Page_410_WorkStation_Axis3;
Page_420_WorkStation_ToolDia;
Page_430_WorkStation_Prism;
Page_460_WorkStation_ErrorList;
Page_470_WorkStation_Parameter3;
END_FUNCTION_BLOCK
ACTION Page_000_Start:
(* QVis page 0, start page *)
iIndexPage:=0;
iPageNumber:=iPageNumber+1;
T_Visu.T_PageIndex[iIndexPage].iIndexConfigPage:=iPageNumber;
ptrConfigPage:=ADR(T_Visu.T_ConfigPage[T_Visu.T_PageIndex[iIndexPage].iIndexConfigPage]);
ptrConfigPage^.sName:='Start page';
ptrConfigPage^.wMaskBtPanelLeft:=16#0;
ptrConfigPage^.wMaskBtPanelRight:=16#0;
ptrConfigPage^.wMaskFunctionPanel:=16#0;
(* Navigation panel restriction *)
ptrConfigPage^.wMaskTouchScreenNavPanel:=16#0;
(* Active machine movement mask *)
ptrConfigPage^.wMaskActiveMachineBtPanelLeft:=16#0;
ptrConfigPage^.wMaskActiveMachineBtPanelRight:=16#0;
ptrConfigPage^.wMaskActiveMachineFunctionPanel:=16#0;
ptrConfigPage^.wMaskActiveMachineNavPanel:=16#0;
(* Button edge action *)
ptrConfigPage^.aiRTrigActionPanelRight[1]:=0;
ptrConfigPage^.aiRTrigActionPanelRight[2]:=0;
ptrConfigPage^.aiRTrigActionPanelRight[3]:=0;
ptrConfigPage^.aiRTrigActionPanelRight[4]:=0;
ptrConfigPage^.aiRTrigActionPanelRight[5]:=0;
ptrConfigPage^.aiFTrigActionPanelRight[1]:=0;
ptrConfigPage^.aiFTrigActionPanelRight[2]:=0;
ptrConfigPage^.aiFTrigActionPanelRight[3]:=0;
ptrConfigPage^.aiFTrigActionPanelRight[4]:=0;
ptrConfigPage^.aiFTrigActionPanelRight[5]:=0;
ptrConfigPage^.aiDelayActionPanelRight[1]:=0;
ptrConfigPage^.aiDelayActionPanelRight[2]:=0;
ptrConfigPage^.aiDelayActionPanelRight[3]:=0;
ptrConfigPage^.aiDelayActionPanelRight[4]:=0;
ptrConfigPage^.aiDelayActionPanelRight[5]:=0;
ptrConfigPage^.aiRTrigActionFunctionPanel[1]:=0;
ptrConfigPage^.aiRTrigActionFunctionPanel[2]:=0;
ptrConfigPage^.aiRTrigActionFunctionPanel[3]:=0;
ptrConfigPage^.aiRTrigActionFunctionPanel[4]:=0;
ptrConfigPage^.aiRTrigActionFunctionPanel[5]:=0;
ptrConfigPage^.aiRTrigActionFunctionPanel[6]:=0;
ptrConfigPage^.aiRTrigActionFunctionPanel[7]:=0;
ptrConfigPage^.aiRTrigActionFunctionPanel[8]:=0;
ptrConfigPage^.aiRTrigActionFunctionPanel[9]:=0;
ptrConfigPage^.aiRTrigActionFunctionPanel[10]:=0;
ptrConfigPage^.aiRTrigActionFunctionPanel[11]:=0;
ptrConfigPage^.aiRTrigActionFunctionPanel[12]:=0;
ptrConfigPage^.aiFTrigActionTouchScreenNavPanel[1]:=0;
ptrConfigPage^.aiFTrigActionTouchScreenNavPanel[2]:=0;
ptrConfigPage^.aiFTrigActionTouchScreenNavPanel[3]:=0;
ptrConfigPage^.aiFTrigActionTouchScreenNavPanel[4]:=0;
ptrConfigPage^.aiFTrigActionTouchScreenNavPanel[5]:=0;
ptrConfigPage^.aiFTrigActionTouchScreenNavPanel[6]:=0;
ptrConfigPage^.xMaskBtStart:=TRUE;
ptrConfigPage^.xMaskBtStop:=FALSE;
END_ACTION
ACTION Page_001_BIOS:
(* QVis page 1, BIOS Password StartUp *)
iIndexPage:=1;
iPageNumber:=iPageNumber+1;
T_Visu.T_PageIndex[iIndexPage].iIndexConfigPage:=iPageNumber;
ptrConfigPage:=ADR(T_Visu.T_ConfigPage[T_Visu.T_PageIndex[iIndexPage].iIndexConfigPage]);
ptrConfigPage^.sName:='BIOS Password StartUp';
ptrConfigPage^.wMaskBtPanelLeft:=16#0;
ptrConfigPage^.wMaskBtPanelRight:=16#0;
ptrConfigPage^.wMaskFunctionPanel:=16#0;
(* Navigation panel restriction *)
ptrConfigPage^.wMaskTouchScreenNavPanel:=16#0;
(* Active machine movement mask *)
ptrConfigPage^.wMaskActiveMachineBtPanelLeft:=16#0;
ptrConfigPage^.wMaskActiveMachineBtPanelRight:=16#0;
ptrConfigPage^.wMaskActiveMachineFunctionPanel:=16#0;
ptrConfigPage^.wMaskActiveMachineNavPanel:=16#0;
(* Button edge action *)
ptrConfigPage^.aiRTrigActionPanelRight[1]:=0;
ptrConfigPage^.aiRTrigActionPanelRight[2]:=0;
ptrConfigPage^.aiRTrigActionPanelRight[3]:=0;
ptrConfigPage^.aiRTrigActionPanelRight[4]:=0;
ptrConfigPage^.aiRTrigActionPanelRight[5]:=0;
ptrConfigPage^.aiFTrigActionPanelRight[1]:=0;
ptrConfigPage^.aiFTrigActionPanelRight[2]:=0;
ptrConfigPage^.aiFTrigActionPanelRight[3]:=0;
ptrConfigPage^.aiFTrigActionPanelRight[4]:=0;
ptrConfigPage^.aiFTrigActionPanelRight[5]:=0;
ptrConfigPage^.aiDelayActionPanelRight[1]:=0;
ptrConfigPage^.aiDelayActionPanelRight[2]:=0;
ptrConfigPage^.aiDelayActionPanelRight[3]:=0;
ptrConfigPage^.aiDelayActionPanelRight[4]:=0;
ptrConfigPage^.aiDelayActionPanelRight[5]:=0;
ptrConfigPage^.aiRTrigActionFunctionPanel[1]:=0;
ptrConfigPage^.aiRTrigActionFunctionPanel[2]:=0;
ptrConfigPage^.aiRTrigActionFunctionPanel[3]:=0;
ptrConfigPage^.aiRTrigActionFunctionPanel[4]:=0;
ptrConfigPage^.aiRTrigActionFunctionPanel[5]:=0;
ptrConfigPage^.aiRTrigActionFunctionPanel[6]:=0;
ptrConfigPage^.aiRTrigActionFunctionPanel[7]:=0;
ptrConfigPage^.aiRTrigActionFunctionPanel[8]:=0;
ptrConfigPage^.aiRTrigActionFunctionPanel[9]:=0;
ptrConfigPage^.aiRTrigActionFunctionPanel[10]:=0;
ptrConfigPage^.aiRTrigActionFunctionPanel[11]:=0;
ptrConfigPage^.aiRTrigActionFunctionPanel[12]:=0;
ptrConfigPage^.aiFTrigActionTouchScreenNavPanel[1]:=0;
ptrConfigPage^.aiFTrigActionTouchScreenNavPanel[2]:=0;
ptrConfigPage^.aiFTrigActionTouchScreenNavPanel[3]:=0;
ptrConfigPage^.aiFTrigActionTouchScreenNavPanel[4]:=0;
ptrConfigPage^.aiFTrigActionTouchScreenNavPanel[5]:=0;
ptrConfigPage^.aiFTrigActionTouchScreenNavPanel[6]:=0;
ptrConfigPage^.xMaskBtStart:=FALSE;
ptrConfigPage^.xMaskBtStop:=FALSE;
END_ACTION
ACTION Page_002_BIOS:
(* QVis page 2, BIOS Parameter StartUp *)
iIndexPage:=2;
iPageNumber:=iPageNumber+1;
T_Visu.T_PageIndex[iIndexPage].iIndexConfigPage:=iPageNumber;
ptrConfigPage:=ADR(T_Visu.T_ConfigPage[T_Visu.T_PageIndex[iIndexPage].iIndexConfigPage]);
ptrConfigPage^.sName:='BIOS Parameter StartUp';
ptrConfigPage^.wMaskBtPanelLeft:=16#0;
ptrConfigPage^.wMaskBtPanelRight:=16#200;
ptrConfigPage^.wMaskFunctionPanel:=16#0;
(* Navigation panel restriction *)
ptrConfigPage^.wMaskTouchScreenNavPanel:=16#0;
(* Active machine movement mask *)
ptrConfigPage^.wMaskActiveMachineBtPanelLeft:=16#0;
ptrConfigPage^.wMaskActiveMachineBtPanelRight:=16#200;
ptrConfigPage^.wMaskActiveMachineFunctionPanel:=16#0;
ptrConfigPage^.wMaskActiveMachineNavPanel:=16#0;
(* Button edge action *)
ptrConfigPage^.aiRTrigActionPanelRight[1]:=0;
ptrConfigPage^.aiRTrigActionPanelRight[2]:=0;
ptrConfigPage^.aiRTrigActionPanelRight[3]:=0;
ptrConfigPage^.aiRTrigActionPanelRight[4]:=0;
ptrConfigPage^.aiRTrigActionPanelRight[5]:=0;
ptrConfigPage^.aiFTrigActionPanelRight[1]:=0;
ptrConfigPage^.aiFTrigActionPanelRight[2]:=0;
ptrConfigPage^.aiFTrigActionPanelRight[3]:=0;
ptrConfigPage^.aiFTrigActionPanelRight[4]:=0;
ptrConfigPage^.aiFTrigActionPanelRight[5]:=0;
ptrConfigPage^.aiDelayActionPanelRight[1]:=0;
ptrConfigPage^.aiDelayActionPanelRight[2]:=0;
ptrConfigPage^.aiDelayActionPanelRight[3]:=0;
ptrConfigPage^.aiDelayActionPanelRight[4]:=0;
ptrConfigPage^.aiDelayActionPanelRight[5]:=0;
ptrConfigPage^.aiRTrigActionFunctionPanel[1]:=0;
ptrConfigPage^.aiRTrigActionFunctionPanel[2]:=0;
ptrConfigPage^.aiRTrigActionFunctionPanel[3]:=0;
ptrConfigPage^.aiRTrigActionFunctionPanel[4]:=0;
ptrConfigPage^.aiRTrigActionFunctionPanel[5]:=0;
ptrConfigPage^.aiRTrigActionFunctionPanel[6]:=0;
ptrConfigPage^.aiRTrigActionFunctionPanel[7]:=0;
ptrConfigPage^.aiRTrigActionFunctionPanel[8]:=0;
ptrConfigPage^.aiRTrigActionFunctionPanel[9]:=0;
ptrConfigPage^.aiRTrigActionFunctionPanel[10]:=0;
ptrConfigPage^.aiRTrigActionFunctionPanel[11]:=0;
ptrConfigPage^.aiRTrigActionFunctionPanel[12]:=0;
ptrConfigPage^.aiFTrigActionTouchScreenNavPanel[1]:=0;
ptrConfigPage^.aiFTrigActionTouchScreenNavPanel[2]:=0;
ptrConfigPage^.aiFTrigActionTouchScreenNavPanel[3]:=0;
ptrConfigPage^.aiFTrigActionTouchScreenNavPanel[4]:=0;
ptrConfigPage^.aiFTrigActionTouchScreenNavPanel[5]:=0;
ptrConfigPage^.aiFTrigActionTouchScreenNavPanel[6]:=0;
ptrConfigPage^.xMaskBtStart:=FALSE;
ptrConfigPage^.xMaskBtStop:=FALSE;
END_ACTION
ACTION Page_010_Auto_Geometry1:
(* QVis page 10, Auto Geometry, page 1 *)
iIndexPage:=10;
iPageNumber:=iPageNumber+1;
T_Visu.T_PageIndex[iIndexPage].iIndexConfigPage:=iPageNumber;
ptrConfigPage:=ADR(T_Visu.T_ConfigPage[T_Visu.T_PageIndex[iIndexPage].iIndexConfigPage]);
ptrConfigPage^.sName:='Auto Geometry, page 1';
ptrConfigPage^.wMaskBtPanelLeft:=16#F;
ptrConfigPage^.wMaskBtPanelRight:=16#200;
(*08.07.2014: KFS	{	*)
(*ptrConfigPage^.wMaskFunctionPanel:=16#F;*)
ptrConfigPage^.wMaskFunctionPanel:=16#3F;
(*08.07.2014: KFS	}	*)
(* Navigation panel restriction *)
ptrConfigPage^.wMaskTouchScreenNavPanel:=16#3F;
(* Active machine movement mask *)
ptrConfigPage^.wMaskActiveMachineBtPanelLeft:=16#F;
ptrConfigPage^.wMaskActiveMachineBtPanelRight:=16#220;
ptrConfigPage^.wMaskActiveMachineFunctionPanel:=16#0;
ptrConfigPage^.wMaskActiveMachineNavPanel:=16#3F;
(* Button edge action *)
ptrConfigPage^.aiRTrigActionPanelRight[1]:=801;
ptrConfigPage^.aiRTrigActionPanelRight[2]:=0;
ptrConfigPage^.aiRTrigActionPanelRight[3]:=0;
ptrConfigPage^.aiRTrigActionPanelRight[4]:=0;
ptrConfigPage^.aiRTrigActionPanelRight[5]:=12;
ptrConfigPage^.aiFTrigActionPanelRight[1]:=0;
ptrConfigPage^.aiFTrigActionPanelRight[2]:=0;
ptrConfigPage^.aiFTrigActionPanelRight[3]:=0;
ptrConfigPage^.aiFTrigActionPanelRight[4]:=0;
ptrConfigPage^.aiFTrigActionPanelRight[5]:=0;
ptrConfigPage^.aiDelayActionPanelRight[1]:=0;
ptrConfigPage^.aiDelayActionPanelRight[2]:=0;
ptrConfigPage^.aiDelayActionPanelRight[3]:=0;
ptrConfigPage^.aiDelayActionPanelRight[4]:=0;
ptrConfigPage^.aiDelayActionPanelRight[5]:=0;
ptrConfigPage^.aiRTrigActionFunctionPanel[1]:=102;
ptrConfigPage^.aiRTrigActionFunctionPanel[2]:=103;
ptrConfigPage^.aiRTrigActionFunctionPanel[3]:=501;
ptrConfigPage^.aiRTrigActionFunctionPanel[4]:=106;
ptrConfigPage^.aiRTrigActionFunctionPanel[5]:=107;
ptrConfigPage^.aiRTrigActionFunctionPanel[6]:=108;
ptrConfigPage^.aiRTrigActionFunctionPanel[7]:=0;
ptrConfigPage^.aiRTrigActionFunctionPanel[8]:=0;
ptrConfigPage^.aiRTrigActionFunctionPanel[9]:=0;
ptrConfigPage^.aiRTrigActionFunctionPanel[10]:=0;
ptrConfigPage^.aiRTrigActionFunctionPanel[11]:=0;
ptrConfigPage^.aiRTrigActionFunctionPanel[12]:=0;
ptrConfigPage^.aiFTrigActionTouchScreenNavPanel[1]:=10010;
ptrConfigPage^.aiFTrigActionTouchScreenNavPanel[2]:=10020;
ptrConfigPage^.aiFTrigActionTouchScreenNavPanel[3]:=10030;
ptrConfigPage^.aiFTrigActionTouchScreenNavPanel[4]:=10040;
ptrConfigPage^.aiFTrigActionTouchScreenNavPanel[5]:=10050;
ptrConfigPage^.aiFTrigActionTouchScreenNavPanel[6]:=10060;
ptrConfigPage^.xMaskBtStart:=TRUE;
ptrConfigPage^.xMaskBtStop:=TRUE;
END_ACTION
ACTION Page_011_Auto_Geometry2:
(* QVis page 11, Auto Geometry, page 2 *)
iIndexPage:=11;
iPageNumber:=iPageNumber+1;
T_Visu.T_PageIndex[iIndexPage].iIndexConfigPage:=iPageNumber;
ptrConfigPage:=ADR(T_Visu.T_ConfigPage[T_Visu.T_PageIndex[iIndexPage].iIndexConfigPage]);
ptrConfigPage^.sName:='Auto Geometry, page 2';
ptrConfigPage^.wMaskBtPanelLeft:=16#F;
ptrConfigPage^.wMaskBtPanelRight:=16#200;
ptrConfigPage^.wMaskFunctionPanel:=16#EF;
(* Navigation panel restriction *)
ptrConfigPage^.wMaskTouchScreenNavPanel:=16#3F;
(* Active machine movement mask *)
ptrConfigPage^.wMaskActiveMachineBtPanelLeft:=16#0;
ptrConfigPage^.wMaskActiveMachineBtPanelRight:=16#0;
ptrConfigPage^.wMaskActiveMachineFunctionPanel:=16#0;
ptrConfigPage^.wMaskActiveMachineNavPanel:=16#3F;
(* Button edge action *)
ptrConfigPage^.aiRTrigActionPanelRight[1]:=0;
ptrConfigPage^.aiRTrigActionPanelRight[2]:=0;
ptrConfigPage^.aiRTrigActionPanelRight[3]:=0;
ptrConfigPage^.aiRTrigActionPanelRight[4]:=0;
ptrConfigPage^.aiRTrigActionPanelRight[5]:=12;
ptrConfigPage^.aiFTrigActionPanelRight[1]:=0;
ptrConfigPage^.aiFTrigActionPanelRight[2]:=0;
ptrConfigPage^.aiFTrigActionPanelRight[3]:=0;
ptrConfigPage^.aiFTrigActionPanelRight[4]:=0;
ptrConfigPage^.aiFTrigActionPanelRight[5]:=0;
ptrConfigPage^.aiDelayActionPanelRight[1]:=0;
ptrConfigPage^.aiDelayActionPanelRight[2]:=0;
ptrConfigPage^.aiDelayActionPanelRight[3]:=0;
ptrConfigPage^.aiDelayActionPanelRight[4]:=0;
ptrConfigPage^.aiDelayActionPanelRight[5]:=0;
ptrConfigPage^.aiRTrigActionFunctionPanel[1]:=110;
ptrConfigPage^.aiRTrigActionFunctionPanel[2]:=111;
ptrConfigPage^.aiRTrigActionFunctionPanel[3]:=114;
ptrConfigPage^.aiRTrigActionFunctionPanel[4]:=115;
ptrConfigPage^.aiRTrigActionFunctionPanel[5]:=0;
ptrConfigPage^.aiRTrigActionFunctionPanel[6]:=116;
ptrConfigPage^.aiRTrigActionFunctionPanel[7]:=112;
ptrConfigPage^.aiRTrigActionFunctionPanel[8]:=113;
ptrConfigPage^.aiRTrigActionFunctionPanel[9]:=0;
ptrConfigPage^.aiRTrigActionFunctionPanel[10]:=0;
ptrConfigPage^.aiRTrigActionFunctionPanel[11]:=0;
ptrConfigPage^.aiRTrigActionFunctionPanel[12]:=0;
ptrConfigPage^.aiFTrigActionTouchScreenNavPanel[1]:=10010;
ptrConfigPage^.aiFTrigActionTouchScreenNavPanel[2]:=10020;
ptrConfigPage^.aiFTrigActionTouchScreenNavPanel[3]:=10030;
ptrConfigPage^.aiFTrigActionTouchScreenNavPanel[4]:=10040;
ptrConfigPage^.aiFTrigActionTouchScreenNavPanel[5]:=10050;
ptrConfigPage^.aiFTrigActionTouchScreenNavPanel[6]:=10060;
ptrConfigPage^.xMaskBtStart:=TRUE;
ptrConfigPage^.xMaskBtStop:=TRUE;
END_ACTION
ACTION Page_020_Auto_Groove1:
(* QVis page 20, Auto Groove, page 1 *)
iIndexPage:=20;
iPageNumber:=iPageNumber+1;
T_Visu.T_PageIndex[iIndexPage].iIndexConfigPage:=iPageNumber;
ptrConfigPage:=ADR(T_Visu.T_ConfigPage[T_Visu.T_PageIndex[iIndexPage].iIndexConfigPage]);
ptrConfigPage^.sName:='Auto Groove, page 1';
ptrConfigPage^.wMaskBtPanelLeft:=16#F;
ptrConfigPage^.wMaskBtPanelRight:=16#200;
ptrConfigPage^.wMaskFunctionPanel:=16#3F;
(* Navigation panel restriction *)
ptrConfigPage^.wMaskTouchScreenNavPanel:=16#3F;
(* Active machine movement mask *)
ptrConfigPage^.wMaskActiveMachineBtPanelLeft:=16#F;
ptrConfigPage^.wMaskActiveMachineBtPanelRight:=16#200;
ptrConfigPage^.wMaskActiveMachineFunctionPanel:=16#0;
ptrConfigPage^.wMaskActiveMachineNavPanel:=16#3F;
(* Button edge action *)
ptrConfigPage^.aiRTrigActionPanelRight[1]:=0;
ptrConfigPage^.aiRTrigActionPanelRight[2]:=0;
ptrConfigPage^.aiRTrigActionPanelRight[3]:=0;
ptrConfigPage^.aiRTrigActionPanelRight[4]:=0;
ptrConfigPage^.aiRTrigActionPanelRight[5]:=12;
ptrConfigPage^.aiFTrigActionPanelRight[1]:=0;
ptrConfigPage^.aiFTrigActionPanelRight[2]:=0;
ptrConfigPage^.aiFTrigActionPanelRight[3]:=0;
ptrConfigPage^.aiFTrigActionPanelRight[4]:=0;
ptrConfigPage^.aiFTrigActionPanelRight[5]:=0;
ptrConfigPage^.aiDelayActionPanelRight[1]:=0;
ptrConfigPage^.aiDelayActionPanelRight[2]:=0;
ptrConfigPage^.aiDelayActionPanelRight[3]:=0;
ptrConfigPage^.aiDelayActionPanelRight[4]:=0;
ptrConfigPage^.aiDelayActionPanelRight[5]:=0;
ptrConfigPage^.aiRTrigActionFunctionPanel[1]:=102;
ptrConfigPage^.aiRTrigActionFunctionPanel[2]:=103;
ptrConfigPage^.aiRTrigActionFunctionPanel[3]:=501;
ptrConfigPage^.aiRTrigActionFunctionPanel[4]:=105;
ptrConfigPage^.aiRTrigActionFunctionPanel[5]:=107;
ptrConfigPage^.aiRTrigActionFunctionPanel[6]:=104;
ptrConfigPage^.aiRTrigActionFunctionPanel[7]:=0;
ptrConfigPage^.aiRTrigActionFunctionPanel[8]:=0;
ptrConfigPage^.aiRTrigActionFunctionPanel[9]:=0;
ptrConfigPage^.aiRTrigActionFunctionPanel[10]:=0;
ptrConfigPage^.aiRTrigActionFunctionPanel[11]:=0;
ptrConfigPage^.aiRTrigActionFunctionPanel[12]:=0;
ptrConfigPage^.aiFTrigActionTouchScreenNavPanel[1]:=10010;
ptrConfigPage^.aiFTrigActionTouchScreenNavPanel[2]:=10020;
ptrConfigPage^.aiFTrigActionTouchScreenNavPanel[3]:=10030;
ptrConfigPage^.aiFTrigActionTouchScreenNavPanel[4]:=10040;
ptrConfigPage^.aiFTrigActionTouchScreenNavPanel[5]:=10050;
ptrConfigPage^.aiFTrigActionTouchScreenNavPanel[6]:=10060;
ptrConfigPage^.xMaskBtStart:=TRUE;
ptrConfigPage^.xMaskBtStop:=TRUE;
END_ACTION
ACTION Page_021_Auto_Groove2:
(* QVis page 21, Auto Groove, page 2 *)
iIndexPage:=21;
iPageNumber:=iPageNumber+1;
T_Visu.T_PageIndex[iIndexPage].iIndexConfigPage:=iPageNumber;
ptrConfigPage:=ADR(T_Visu.T_ConfigPage[T_Visu.T_PageIndex[iIndexPage].iIndexConfigPage]);
ptrConfigPage^.sName:='Auto Groove, page 2';
ptrConfigPage^.wMaskBtPanelLeft:=16#F;
ptrConfigPage^.wMaskBtPanelRight:=16#200;
ptrConfigPage^.wMaskFunctionPanel:=16#EF;
(* Navigation panel restriction *)
ptrConfigPage^.wMaskTouchScreenNavPanel:=16#3F;
(* Active machine movement mask *)
ptrConfigPage^.wMaskActiveMachineBtPanelLeft:=16#0;
ptrConfigPage^.wMaskActiveMachineBtPanelRight:=16#0;
ptrConfigPage^.wMaskActiveMachineFunctionPanel:=16#0;
ptrConfigPage^.wMaskActiveMachineNavPanel:=16#3F;
(* Button edge action *)
ptrConfigPage^.aiRTrigActionPanelRight[1]:=0;
ptrConfigPage^.aiRTrigActionPanelRight[2]:=0;
ptrConfigPage^.aiRTrigActionPanelRight[3]:=0;
ptrConfigPage^.aiRTrigActionPanelRight[4]:=0;
ptrConfigPage^.aiRTrigActionPanelRight[5]:=12;
ptrConfigPage^.aiFTrigActionPanelRight[1]:=0;
ptrConfigPage^.aiFTrigActionPanelRight[2]:=0;
ptrConfigPage^.aiFTrigActionPanelRight[3]:=0;
ptrConfigPage^.aiFTrigActionPanelRight[4]:=0;
ptrConfigPage^.aiFTrigActionPanelRight[5]:=0;
ptrConfigPage^.aiDelayActionPanelRight[1]:=0;
ptrConfigPage^.aiDelayActionPanelRight[2]:=0;
ptrConfigPage^.aiDelayActionPanelRight[3]:=0;
ptrConfigPage^.aiDelayActionPanelRight[4]:=0;
ptrConfigPage^.aiDelayActionPanelRight[5]:=0;
ptrConfigPage^.aiRTrigActionFunctionPanel[1]:=110;
ptrConfigPage^.aiRTrigActionFunctionPanel[2]:=111;
ptrConfigPage^.aiRTrigActionFunctionPanel[3]:=114;
ptrConfigPage^.aiRTrigActionFunctionPanel[4]:=115;
ptrConfigPage^.aiRTrigActionFunctionPanel[5]:=0;
ptrConfigPage^.aiRTrigActionFunctionPanel[6]:=116;
ptrConfigPage^.aiRTrigActionFunctionPanel[7]:=112;
ptrConfigPage^.aiRTrigActionFunctionPanel[8]:=113;
ptrConfigPage^.aiRTrigActionFunctionPanel[9]:=0;
ptrConfigPage^.aiRTrigActionFunctionPanel[10]:=0;
ptrConfigPage^.aiRTrigActionFunctionPanel[11]:=0;
ptrConfigPage^.aiRTrigActionFunctionPanel[12]:=0;
ptrConfigPage^.aiFTrigActionTouchScreenNavPanel[1]:=10010;
ptrConfigPage^.aiFTrigActionTouchScreenNavPanel[2]:=10020;
ptrConfigPage^.aiFTrigActionTouchScreenNavPanel[3]:=10030;
ptrConfigPage^.aiFTrigActionTouchScreenNavPanel[4]:=10040;
ptrConfigPage^.aiFTrigActionTouchScreenNavPanel[5]:=10050;
ptrConfigPage^.aiFTrigActionTouchScreenNavPanel[6]:=10060;
ptrConfigPage^.xMaskBtStart:=TRUE;
ptrConfigPage^.xMaskBtStop:=TRUE;
END_ACTION
ACTION Page_030_Auto_Reference:
(* QVis page 30, Reference *)
iIndexPage:=30;
iPageNumber:=iPageNumber+1;
T_Visu.T_PageIndex[iIndexPage].iIndexConfigPage:=iPageNumber;
ptrConfigPage:=ADR(T_Visu.T_ConfigPage[T_Visu.T_PageIndex[iIndexPage].iIndexConfigPage]);
ptrConfigPage^.sName:='Reference';
ptrConfigPage^.wMaskBtPanelLeft:=16#F;
ptrConfigPage^.wMaskBtPanelRight:=16#1E0;
ptrConfigPage^.wMaskFunctionPanel:=16#D;
(* Navigation panel restriction *)
ptrConfigPage^.wMaskTouchScreenNavPanel:=16#3F;
(* Active machine movement mask *)
ptrConfigPage^.wMaskActiveMachineBtPanelLeft:=16#F;
ptrConfigPage^.wMaskActiveMachineBtPanelRight:=16#60;
ptrConfigPage^.wMaskActiveMachineFunctionPanel:=16#0;
ptrConfigPage^.wMaskActiveMachineNavPanel:=16#3F;
(* Button edge action *)
ptrConfigPage^.aiRTrigActionPanelRight[1]:=312;
ptrConfigPage^.aiRTrigActionPanelRight[2]:=310;
ptrConfigPage^.aiRTrigActionPanelRight[3]:=316;
ptrConfigPage^.aiRTrigActionPanelRight[4]:=314;
ptrConfigPage^.aiRTrigActionPanelRight[5]:=0;
ptrConfigPage^.aiFTrigActionPanelRight[1]:=0;
ptrConfigPage^.aiFTrigActionPanelRight[2]:=0;
ptrConfigPage^.aiFTrigActionPanelRight[3]:=301;
ptrConfigPage^.aiFTrigActionPanelRight[4]:=301;
ptrConfigPage^.aiFTrigActionPanelRight[5]:=0;
ptrConfigPage^.aiDelayActionPanelRight[1]:=0;
ptrConfigPage^.aiDelayActionPanelRight[2]:=0;
ptrConfigPage^.aiDelayActionPanelRight[3]:=0;
ptrConfigPage^.aiDelayActionPanelRight[4]:=0;
ptrConfigPage^.aiDelayActionPanelRight[5]:=0;
ptrConfigPage^.aiRTrigActionFunctionPanel[1]:=320;
ptrConfigPage^.aiRTrigActionFunctionPanel[2]:=0;
ptrConfigPage^.aiRTrigActionFunctionPanel[3]:=501;
ptrConfigPage^.aiRTrigActionFunctionPanel[4]:=106;
ptrConfigPage^.aiRTrigActionFunctionPanel[5]:=0;
ptrConfigPage^.aiRTrigActionFunctionPanel[6]:=0;
ptrConfigPage^.aiRTrigActionFunctionPanel[7]:=0;
ptrConfigPage^.aiRTrigActionFunctionPanel[8]:=0;
ptrConfigPage^.aiRTrigActionFunctionPanel[9]:=0;
ptrConfigPage^.aiRTrigActionFunctionPanel[10]:=0;
ptrConfigPage^.aiRTrigActionFunctionPanel[11]:=0;
ptrConfigPage^.aiRTrigActionFunctionPanel[12]:=0;
ptrConfigPage^.aiFTrigActionTouchScreenNavPanel[1]:=10010;
ptrConfigPage^.aiFTrigActionTouchScreenNavPanel[2]:=10020;
ptrConfigPage^.aiFTrigActionTouchScreenNavPanel[3]:=10030;
ptrConfigPage^.aiFTrigActionTouchScreenNavPanel[4]:=10040;
ptrConfigPage^.aiFTrigActionTouchScreenNavPanel[5]:=10050;
ptrConfigPage^.aiFTrigActionTouchScreenNavPanel[6]:=10060;
ptrConfigPage^.xMaskBtStart:=TRUE;
ptrConfigPage^.xMaskBtStop:=TRUE;
END_ACTION
ACTION Page_040_Auto_Setup1:
(* QVis page 40, Setup --> change user level *)
iIndexPage:=40;
iPageNumber:=iPageNumber+1;
T_Visu.T_PageIndex[iIndexPage].iIndexConfigPage:=iPageNumber;
ptrConfigPage:=ADR(T_Visu.T_ConfigPage[T_Visu.T_PageIndex[iIndexPage].iIndexConfigPage]);
ptrConfigPage^.sName:='Setup --> change user level';
ptrConfigPage^.wMaskBtPanelLeft:=16#F;
ptrConfigPage^.wMaskBtPanelRight:=16#200;
ptrConfigPage^.wMaskFunctionPanel:=16#0;
(* Navigation panel restriction *)
ptrConfigPage^.wMaskTouchScreenNavPanel:=16#3F;
(* Active machine movement mask *)
ptrConfigPage^.wMaskActiveMachineBtPanelLeft:=16#0;
ptrConfigPage^.wMaskActiveMachineBtPanelRight:=16#200;
ptrConfigPage^.wMaskActiveMachineFunctionPanel:=16#0;
ptrConfigPage^.wMaskActiveMachineNavPanel:=16#3F;
(* Button edge action *)
ptrConfigPage^.aiRTrigActionPanelRight[1]:=0;
ptrConfigPage^.aiRTrigActionPanelRight[2]:=0;
ptrConfigPage^.aiRTrigActionPanelRight[3]:=0;
ptrConfigPage^.aiRTrigActionPanelRight[4]:=0;
ptrConfigPage^.aiRTrigActionPanelRight[5]:=12;
ptrConfigPage^.aiFTrigActionPanelRight[1]:=0;
ptrConfigPage^.aiFTrigActionPanelRight[2]:=0;
ptrConfigPage^.aiFTrigActionPanelRight[3]:=0;
ptrConfigPage^.aiFTrigActionPanelRight[4]:=0;
ptrConfigPage^.aiFTrigActionPanelRight[5]:=0;
ptrConfigPage^.aiDelayActionPanelRight[1]:=0;
ptrConfigPage^.aiDelayActionPanelRight[2]:=0;
ptrConfigPage^.aiDelayActionPanelRight[3]:=0;
ptrConfigPage^.aiDelayActionPanelRight[4]:=0;
ptrConfigPage^.aiDelayActionPanelRight[5]:=0;
ptrConfigPage^.aiRTrigActionFunctionPanel[1]:=0;
ptrConfigPage^.aiRTrigActionFunctionPanel[2]:=0;
ptrConfigPage^.aiRTrigActionFunctionPanel[3]:=0;
ptrConfigPage^.aiRTrigActionFunctionPanel[4]:=0;
ptrConfigPage^.aiRTrigActionFunctionPanel[5]:=0;
ptrConfigPage^.aiRTrigActionFunctionPanel[6]:=0;
ptrConfigPage^.aiRTrigActionFunctionPanel[7]:=0;
ptrConfigPage^.aiRTrigActionFunctionPanel[8]:=0;
ptrConfigPage^.aiRTrigActionFunctionPanel[9]:=0;
ptrConfigPage^.aiRTrigActionFunctionPanel[10]:=0;
ptrConfigPage^.aiRTrigActionFunctionPanel[11]:=0;
ptrConfigPage^.aiRTrigActionFunctionPanel[12]:=0;
ptrConfigPage^.aiFTrigActionTouchScreenNavPanel[1]:=10010;
ptrConfigPage^.aiFTrigActionTouchScreenNavPanel[2]:=10020;
ptrConfigPage^.aiFTrigActionTouchScreenNavPanel[3]:=10030;
ptrConfigPage^.aiFTrigActionTouchScreenNavPanel[4]:=10040;
ptrConfigPage^.aiFTrigActionTouchScreenNavPanel[5]:=10050;
ptrConfigPage^.aiFTrigActionTouchScreenNavPanel[6]:=10060;
ptrConfigPage^.xMaskBtStart:=FALSE;
ptrConfigPage^.xMaskBtStop:=TRUE;
END_ACTION
ACTION Page_041_Auto_Setup2:
(* QVis page 41, Setup --> change language *)
iIndexPage:=41;
iPageNumber:=iPageNumber+1;
T_Visu.T_PageIndex[iIndexPage].iIndexConfigPage:=iPageNumber;
ptrConfigPage:=ADR(T_Visu.T_ConfigPage[T_Visu.T_PageIndex[iIndexPage].iIndexConfigPage]);
ptrConfigPage^.sName:='Setup --> change language';
ptrConfigPage^.wMaskBtPanelLeft:=16#F;
ptrConfigPage^.wMaskBtPanelRight:=16#200;
ptrConfigPage^.wMaskFunctionPanel:=16#0;
(* Navigation panel restriction *)
ptrConfigPage^.wMaskTouchScreenNavPanel:=16#3F;
(* Active machine movement mask *)
ptrConfigPage^.wMaskActiveMachineBtPanelLeft:=16#0;
ptrConfigPage^.wMaskActiveMachineBtPanelRight:=16#200;
ptrConfigPage^.wMaskActiveMachineFunctionPanel:=16#0;
ptrConfigPage^.wMaskActiveMachineNavPanel:=16#3F;
(* Button edge action *)
ptrConfigPage^.aiRTrigActionPanelRight[1]:=0;
ptrConfigPage^.aiRTrigActionPanelRight[2]:=0;
ptrConfigPage^.aiRTrigActionPanelRight[3]:=0;
ptrConfigPage^.aiRTrigActionPanelRight[4]:=0;
ptrConfigPage^.aiRTrigActionPanelRight[5]:=12;
ptrConfigPage^.aiFTrigActionPanelRight[1]:=0;
ptrConfigPage^.aiFTrigActionPanelRight[2]:=0;
ptrConfigPage^.aiFTrigActionPanelRight[3]:=0;
ptrConfigPage^.aiFTrigActionPanelRight[4]:=0;
ptrConfigPage^.aiFTrigActionPanelRight[5]:=0;
ptrConfigPage^.aiDelayActionPanelRight[1]:=0;
ptrConfigPage^.aiDelayActionPanelRight[2]:=0;
ptrConfigPage^.aiDelayActionPanelRight[3]:=0;
ptrConfigPage^.aiDelayActionPanelRight[4]:=0;
ptrConfigPage^.aiDelayActionPanelRight[5]:=0;
ptrConfigPage^.aiRTrigActionFunctionPanel[1]:=0;
ptrConfigPage^.aiRTrigActionFunctionPanel[2]:=0;
ptrConfigPage^.aiRTrigActionFunctionPanel[3]:=0;
ptrConfigPage^.aiRTrigActionFunctionPanel[4]:=0;
ptrConfigPage^.aiRTrigActionFunctionPanel[5]:=0;
ptrConfigPage^.aiRTrigActionFunctionPanel[6]:=0;
ptrConfigPage^.aiRTrigActionFunctionPanel[7]:=0;
ptrConfigPage^.aiRTrigActionFunctionPanel[8]:=0;
ptrConfigPage^.aiRTrigActionFunctionPanel[9]:=0;
ptrConfigPage^.aiRTrigActionFunctionPanel[10]:=0;
ptrConfigPage^.aiRTrigActionFunctionPanel[11]:=0;
ptrConfigPage^.aiRTrigActionFunctionPanel[12]:=0;
ptrConfigPage^.aiFTrigActionTouchScreenNavPanel[1]:=10010;
ptrConfigPage^.aiFTrigActionTouchScreenNavPanel[2]:=10020;
ptrConfigPage^.aiFTrigActionTouchScreenNavPanel[3]:=10030;
ptrConfigPage^.aiFTrigActionTouchScreenNavPanel[4]:=10040;
ptrConfigPage^.aiFTrigActionTouchScreenNavPanel[5]:=10050;
ptrConfigPage^.aiFTrigActionTouchScreenNavPanel[6]:=10060;
ptrConfigPage^.xMaskBtStart:=FALSE;
ptrConfigPage^.xMaskBtStop:=TRUE;
END_ACTION
ACTION Page_050_Auto_Info1:
(* QVis page 50, Axis informations *)
iIndexPage:=50;
iPageNumber:=iPageNumber+1;
T_Visu.T_PageIndex[iIndexPage].iIndexConfigPage:=iPageNumber;
ptrConfigPage:=ADR(T_Visu.T_ConfigPage[T_Visu.T_PageIndex[iIndexPage].iIndexConfigPage]);
ptrConfigPage^.sName:='Axis informations';
ptrConfigPage^.wMaskBtPanelLeft:=16#F;
ptrConfigPage^.wMaskBtPanelRight:=16#200;
ptrConfigPage^.wMaskFunctionPanel:=16#0;
(* Navigation panel restriction *)
ptrConfigPage^.wMaskTouchScreenNavPanel:=16#3F;
(* Active machine movement mask *)
ptrConfigPage^.wMaskActiveMachineBtPanelLeft:=16#0;
ptrConfigPage^.wMaskActiveMachineBtPanelRight:=16#200;
ptrConfigPage^.wMaskActiveMachineFunctionPanel:=16#0;
ptrConfigPage^.wMaskActiveMachineNavPanel:=16#3F;
(* Button edge action *)
ptrConfigPage^.aiRTrigActionPanelRight[1]:=0;
ptrConfigPage^.aiRTrigActionPanelRight[2]:=0;
ptrConfigPage^.aiRTrigActionPanelRight[3]:=0;
ptrConfigPage^.aiRTrigActionPanelRight[4]:=0;
ptrConfigPage^.aiRTrigActionPanelRight[5]:=12;
ptrConfigPage^.aiFTrigActionPanelRight[1]:=0;
ptrConfigPage^.aiFTrigActionPanelRight[2]:=0;
ptrConfigPage^.aiFTrigActionPanelRight[3]:=0;
ptrConfigPage^.aiFTrigActionPanelRight[4]:=0;
ptrConfigPage^.aiFTrigActionPanelRight[5]:=0;
ptrConfigPage^.aiDelayActionPanelRight[1]:=0;
ptrConfigPage^.aiDelayActionPanelRight[2]:=0;
ptrConfigPage^.aiDelayActionPanelRight[3]:=0;
ptrConfigPage^.aiDelayActionPanelRight[4]:=0;
ptrConfigPage^.aiDelayActionPanelRight[5]:=0;
ptrConfigPage^.aiRTrigActionFunctionPanel[1]:=0;
ptrConfigPage^.aiRTrigActionFunctionPanel[2]:=0;
ptrConfigPage^.aiRTrigActionFunctionPanel[3]:=0;
ptrConfigPage^.aiRTrigActionFunctionPanel[4]:=0;
ptrConfigPage^.aiRTrigActionFunctionPanel[5]:=0;
ptrConfigPage^.aiRTrigActionFunctionPanel[6]:=0;
ptrConfigPage^.aiRTrigActionFunctionPanel[7]:=0;
ptrConfigPage^.aiRTrigActionFunctionPanel[8]:=0;
ptrConfigPage^.aiRTrigActionFunctionPanel[9]:=0;
ptrConfigPage^.aiRTrigActionFunctionPanel[10]:=0;
ptrConfigPage^.aiRTrigActionFunctionPanel[11]:=0;
ptrConfigPage^.aiRTrigActionFunctionPanel[12]:=0;
ptrConfigPage^.aiFTrigActionTouchScreenNavPanel[1]:=10010;
ptrConfigPage^.aiFTrigActionTouchScreenNavPanel[2]:=10020;
ptrConfigPage^.aiFTrigActionTouchScreenNavPanel[3]:=10030;
ptrConfigPage^.aiFTrigActionTouchScreenNavPanel[4]:=10040;
ptrConfigPage^.aiFTrigActionTouchScreenNavPanel[5]:=10050;
ptrConfigPage^.aiFTrigActionTouchScreenNavPanel[6]:=10060;
ptrConfigPage^.xMaskBtStart:=FALSE;
ptrConfigPage^.xMaskBtStop:=TRUE;
END_ACTION
ACTION Page_051_Auto_Info2:
(* QVis page 51, System informations *)
iIndexPage:=51;
iPageNumber:=iPageNumber+1;
T_Visu.T_PageIndex[iIndexPage].iIndexConfigPage:=iPageNumber;
ptrConfigPage:=ADR(T_Visu.T_ConfigPage[T_Visu.T_PageIndex[iIndexPage].iIndexConfigPage]);
ptrConfigPage^.sName:='System informations';
ptrConfigPage^.wMaskBtPanelLeft:=16#F;
ptrConfigPage^.wMaskBtPanelRight:=16#200;
ptrConfigPage^.wMaskFunctionPanel:=16#0;
(* Navigation panel restriction *)
ptrConfigPage^.wMaskTouchScreenNavPanel:=16#3F;
(* Active machine movement mask *)
ptrConfigPage^.wMaskActiveMachineBtPanelLeft:=16#0;
ptrConfigPage^.wMaskActiveMachineBtPanelRight:=16#200;
ptrConfigPage^.wMaskActiveMachineFunctionPanel:=16#0;
ptrConfigPage^.wMaskActiveMachineNavPanel:=16#3F;
(* Button edge action *)
ptrConfigPage^.aiRTrigActionPanelRight[1]:=0;
ptrConfigPage^.aiRTrigActionPanelRight[2]:=0;
ptrConfigPage^.aiRTrigActionPanelRight[3]:=0;
ptrConfigPage^.aiRTrigActionPanelRight[4]:=0;
ptrConfigPage^.aiRTrigActionPanelRight[5]:=12;
ptrConfigPage^.aiFTrigActionPanelRight[1]:=0;
ptrConfigPage^.aiFTrigActionPanelRight[2]:=0;
ptrConfigPage^.aiFTrigActionPanelRight[3]:=0;
ptrConfigPage^.aiFTrigActionPanelRight[4]:=0;
ptrConfigPage^.aiFTrigActionPanelRight[5]:=0;
ptrConfigPage^.aiDelayActionPanelRight[1]:=0;
ptrConfigPage^.aiDelayActionPanelRight[2]:=0;
ptrConfigPage^.aiDelayActionPanelRight[3]:=0;
ptrConfigPage^.aiDelayActionPanelRight[4]:=0;
ptrConfigPage^.aiDelayActionPanelRight[5]:=0;
ptrConfigPage^.aiRTrigActionFunctionPanel[1]:=0;
ptrConfigPage^.aiRTrigActionFunctionPanel[2]:=0;
ptrConfigPage^.aiRTrigActionFunctionPanel[3]:=0;
ptrConfigPage^.aiRTrigActionFunctionPanel[4]:=0;
ptrConfigPage^.aiRTrigActionFunctionPanel[5]:=0;
ptrConfigPage^.aiRTrigActionFunctionPanel[6]:=0;
ptrConfigPage^.aiRTrigActionFunctionPanel[7]:=0;
ptrConfigPage^.aiRTrigActionFunctionPanel[8]:=0;
ptrConfigPage^.aiRTrigActionFunctionPanel[9]:=0;
ptrConfigPage^.aiRTrigActionFunctionPanel[10]:=0;
ptrConfigPage^.aiRTrigActionFunctionPanel[11]:=0;
ptrConfigPage^.aiRTrigActionFunctionPanel[12]:=0;
ptrConfigPage^.aiFTrigActionTouchScreenNavPanel[1]:=10010;
ptrConfigPage^.aiFTrigActionTouchScreenNavPanel[2]:=10020;
ptrConfigPage^.aiFTrigActionTouchScreenNavPanel[3]:=10030;
ptrConfigPage^.aiFTrigActionTouchScreenNavPanel[4]:=10040;
ptrConfigPage^.aiFTrigActionTouchScreenNavPanel[5]:=10050;
ptrConfigPage^.aiFTrigActionTouchScreenNavPanel[6]:=10060;
ptrConfigPage^.xMaskBtStart:=FALSE;
ptrConfigPage^.xMaskBtStop:=TRUE;
END_ACTION
ACTION Page_060_Auto_ErrorList:
(* QVis page 60, Error List *)
iIndexPage:=60;
iPageNumber:=iPageNumber+1;
T_Visu.T_PageIndex[iIndexPage].iIndexConfigPage:=iPageNumber;
ptrConfigPage:=ADR(T_Visu.T_ConfigPage[T_Visu.T_PageIndex[iIndexPage].iIndexConfigPage]);
ptrConfigPage^.sName:='Error List';
ptrConfigPage^.wMaskBtPanelLeft:=16#F;
ptrConfigPage^.wMaskBtPanelRight:=16#60;
ptrConfigPage^.wMaskFunctionPanel:=16#0;
(* Navigation panel restriction *)
ptrConfigPage^.wMaskTouchScreenNavPanel:=16#3F;
(* Active machine movement mask *)
ptrConfigPage^.wMaskActiveMachineBtPanelLeft:=16#0;
ptrConfigPage^.wMaskActiveMachineBtPanelRight:=16#60;
ptrConfigPage^.wMaskActiveMachineFunctionPanel:=16#0;
ptrConfigPage^.wMaskActiveMachineNavPanel:=16#3F;
(* Button edge action *)
ptrConfigPage^.aiRTrigActionPanelRight[1]:=99;
ptrConfigPage^.aiRTrigActionPanelRight[2]:=20;
ptrConfigPage^.aiRTrigActionPanelRight[3]:=0;
ptrConfigPage^.aiRTrigActionPanelRight[4]:=0;
ptrConfigPage^.aiRTrigActionPanelRight[5]:=0;
ptrConfigPage^.aiFTrigActionPanelRight[1]:=0;
ptrConfigPage^.aiFTrigActionPanelRight[2]:=0;
ptrConfigPage^.aiFTrigActionPanelRight[3]:=0;
ptrConfigPage^.aiFTrigActionPanelRight[4]:=0;
ptrConfigPage^.aiFTrigActionPanelRight[5]:=0;
ptrConfigPage^.aiDelayActionPanelRight[1]:=0;
ptrConfigPage^.aiDelayActionPanelRight[2]:=0;
ptrConfigPage^.aiDelayActionPanelRight[3]:=0;
ptrConfigPage^.aiDelayActionPanelRight[4]:=0;
ptrConfigPage^.aiDelayActionPanelRight[5]:=0;
ptrConfigPage^.aiRTrigActionFunctionPanel[1]:=0;
ptrConfigPage^.aiRTrigActionFunctionPanel[2]:=0;
ptrConfigPage^.aiRTrigActionFunctionPanel[3]:=0;
ptrConfigPage^.aiRTrigActionFunctionPanel[4]:=0;
ptrConfigPage^.aiRTrigActionFunctionPanel[5]:=0;
ptrConfigPage^.aiRTrigActionFunctionPanel[6]:=0;
ptrConfigPage^.aiRTrigActionFunctionPanel[7]:=0;
ptrConfigPage^.aiRTrigActionFunctionPanel[8]:=0;
ptrConfigPage^.aiRTrigActionFunctionPanel[9]:=0;
ptrConfigPage^.aiRTrigActionFunctionPanel[10]:=0;
ptrConfigPage^.aiRTrigActionFunctionPanel[11]:=0;
ptrConfigPage^.aiRTrigActionFunctionPanel[12]:=0;
ptrConfigPage^.aiFTrigActionTouchScreenNavPanel[1]:=10010;
ptrConfigPage^.aiFTrigActionTouchScreenNavPanel[2]:=10020;
ptrConfigPage^.aiFTrigActionTouchScreenNavPanel[3]:=10030;
ptrConfigPage^.aiFTrigActionTouchScreenNavPanel[4]:=10040;
ptrConfigPage^.aiFTrigActionTouchScreenNavPanel[5]:=10050;
ptrConfigPage^.aiFTrigActionTouchScreenNavPanel[6]:=10060;
ptrConfigPage^.xMaskBtStart:=FALSE;
ptrConfigPage^.xMaskBtStop:=TRUE;
END_ACTION
ACTION Page_110_Setup_ToolCalibration:
(* QVis page 110, Tool Calibration *)
iIndexPage:=110;
iPageNumber:=iPageNumber+1;
T_Visu.T_PageIndex[iIndexPage].iIndexConfigPage:=iPageNumber;
ptrConfigPage:=ADR(T_Visu.T_ConfigPage[T_Visu.T_PageIndex[iIndexPage].iIndexConfigPage]);
ptrConfigPage^.sName:='Tool Calibration';
ptrConfigPage^.wMaskBtPanelLeft:=16#1F;
ptrConfigPage^.wMaskBtPanelRight:=16#0;
ptrConfigPage^.wMaskFunctionPanel:=16#3F;
(* Navigation panel restriction *)
ptrConfigPage^.wMaskTouchScreenNavPanel:=16#3F;
(* Active machine movement mask *)
ptrConfigPage^.wMaskActiveMachineBtPanelLeft:=16#F;
ptrConfigPage^.wMaskActiveMachineBtPanelRight:=16#0;
ptrConfigPage^.wMaskActiveMachineFunctionPanel:=16#0;
ptrConfigPage^.wMaskActiveMachineNavPanel:=16#3F;
(* Button edge action *)
ptrConfigPage^.aiRTrigActionPanelRight[1]:=0;
ptrConfigPage^.aiRTrigActionPanelRight[2]:=0;
ptrConfigPage^.aiRTrigActionPanelRight[3]:=0;
ptrConfigPage^.aiRTrigActionPanelRight[4]:=0;
ptrConfigPage^.aiRTrigActionPanelRight[5]:=0;
ptrConfigPage^.aiFTrigActionPanelRight[1]:=0;
ptrConfigPage^.aiFTrigActionPanelRight[2]:=0;
ptrConfigPage^.aiFTrigActionPanelRight[3]:=0;
ptrConfigPage^.aiFTrigActionPanelRight[4]:=0;
ptrConfigPage^.aiFTrigActionPanelRight[5]:=0;
ptrConfigPage^.aiDelayActionPanelRight[1]:=0;
ptrConfigPage^.aiDelayActionPanelRight[2]:=0;
ptrConfigPage^.aiDelayActionPanelRight[3]:=0;
ptrConfigPage^.aiDelayActionPanelRight[4]:=0;
ptrConfigPage^.aiDelayActionPanelRight[5]:=0;
ptrConfigPage^.aiRTrigActionFunctionPanel[1]:=102;
ptrConfigPage^.aiRTrigActionFunctionPanel[2]:=103;
ptrConfigPage^.aiRTrigActionFunctionPanel[3]:=501;
ptrConfigPage^.aiRTrigActionFunctionPanel[4]:=132;
ptrConfigPage^.aiRTrigActionFunctionPanel[5]:=105;
ptrConfigPage^.aiRTrigActionFunctionPanel[6]:=101;
ptrConfigPage^.aiRTrigActionFunctionPanel[7]:=0;
ptrConfigPage^.aiRTrigActionFunctionPanel[8]:=0;
ptrConfigPage^.aiRTrigActionFunctionPanel[9]:=0;
ptrConfigPage^.aiRTrigActionFunctionPanel[10]:=0;
ptrConfigPage^.aiRTrigActionFunctionPanel[11]:=0;
ptrConfigPage^.aiRTrigActionFunctionPanel[12]:=0;
ptrConfigPage^.aiFTrigActionTouchScreenNavPanel[1]:=10110;
ptrConfigPage^.aiFTrigActionTouchScreenNavPanel[2]:=10120;
ptrConfigPage^.aiFTrigActionTouchScreenNavPanel[3]:=10130;
ptrConfigPage^.aiFTrigActionTouchScreenNavPanel[4]:=10140;
ptrConfigPage^.aiFTrigActionTouchScreenNavPanel[5]:=10150;
ptrConfigPage^.aiFTrigActionTouchScreenNavPanel[6]:=10160;
ptrConfigPage^.xMaskBtStart:=TRUE;
ptrConfigPage^.xMaskBtStop:=TRUE;
END_ACTION
ACTION Page_120_Setup_ToolGeometry1:
(* QVis page 120, Tool Geometry *)
iIndexPage:=120;
iPageNumber:=iPageNumber+1;
T_Visu.T_PageIndex[iIndexPage].iIndexConfigPage:=iPageNumber;
ptrConfigPage:=ADR(T_Visu.T_ConfigPage[T_Visu.T_PageIndex[iIndexPage].iIndexConfigPage]);
ptrConfigPage^.sName:='Tool Geometry';
ptrConfigPage^.wMaskBtPanelLeft:=16#1F;
ptrConfigPage^.wMaskBtPanelRight:=16#60;
ptrConfigPage^.wMaskFunctionPanel:=16#3F;
(* Navigation panel restriction *)
ptrConfigPage^.wMaskTouchScreenNavPanel:=16#3F;
(* Active machine movement mask *)
ptrConfigPage^.wMaskActiveMachineBtPanelLeft:=16#0;
ptrConfigPage^.wMaskActiveMachineBtPanelRight:=16#0;
ptrConfigPage^.wMaskActiveMachineFunctionPanel:=16#0;
ptrConfigPage^.wMaskActiveMachineNavPanel:=16#3F;
(* Button edge action *)
ptrConfigPage^.aiRTrigActionPanelRight[1]:=10120;
ptrConfigPage^.aiRTrigActionPanelRight[2]:=10121;
ptrConfigPage^.aiRTrigActionPanelRight[3]:=0;
ptrConfigPage^.aiRTrigActionPanelRight[4]:=0;
ptrConfigPage^.aiRTrigActionPanelRight[5]:=0;
ptrConfigPage^.aiFTrigActionPanelRight[1]:=0;
ptrConfigPage^.aiFTrigActionPanelRight[2]:=0;
ptrConfigPage^.aiFTrigActionPanelRight[3]:=0;
ptrConfigPage^.aiFTrigActionPanelRight[4]:=0;
ptrConfigPage^.aiFTrigActionPanelRight[5]:=0;
ptrConfigPage^.aiDelayActionPanelRight[1]:=0;
ptrConfigPage^.aiDelayActionPanelRight[2]:=0;
ptrConfigPage^.aiDelayActionPanelRight[3]:=0;
ptrConfigPage^.aiDelayActionPanelRight[4]:=0;
ptrConfigPage^.aiDelayActionPanelRight[5]:=0;
ptrConfigPage^.aiRTrigActionFunctionPanel[1]:=201;
ptrConfigPage^.aiRTrigActionFunctionPanel[2]:=202;
ptrConfigPage^.aiRTrigActionFunctionPanel[3]:=203;
ptrConfigPage^.aiRTrigActionFunctionPanel[4]:=204;
ptrConfigPage^.aiRTrigActionFunctionPanel[5]:=205;
ptrConfigPage^.aiRTrigActionFunctionPanel[6]:=1005;
ptrConfigPage^.aiRTrigActionFunctionPanel[7]:=0;
ptrConfigPage^.aiRTrigActionFunctionPanel[8]:=0;
ptrConfigPage^.aiRTrigActionFunctionPanel[9]:=0;
ptrConfigPage^.aiRTrigActionFunctionPanel[10]:=0;
ptrConfigPage^.aiRTrigActionFunctionPanel[11]:=0;
ptrConfigPage^.aiRTrigActionFunctionPanel[12]:=0;
ptrConfigPage^.aiFTrigActionTouchScreenNavPanel[1]:=10110;
ptrConfigPage^.aiFTrigActionTouchScreenNavPanel[2]:=10120;
ptrConfigPage^.aiFTrigActionTouchScreenNavPanel[3]:=10130;
ptrConfigPage^.aiFTrigActionTouchScreenNavPanel[4]:=10140;
ptrConfigPage^.aiFTrigActionTouchScreenNavPanel[5]:=10150;
ptrConfigPage^.aiFTrigActionTouchScreenNavPanel[6]:=10160;
ptrConfigPage^.xMaskBtStart:=FALSE;
ptrConfigPage^.xMaskBtStop:=TRUE;
END_ACTION
ACTION Page_121_Setup_ToolGeometry2:
(* QVis page 121, Tool Geometry *)
iIndexPage:=121;
iPageNumber:=iPageNumber+1;
T_Visu.T_PageIndex[iIndexPage].iIndexConfigPage:=iPageNumber;
ptrConfigPage:=ADR(T_Visu.T_ConfigPage[T_Visu.T_PageIndex[iIndexPage].iIndexConfigPage]);
ptrConfigPage^.sName:='Tool Geometry';
ptrConfigPage^.wMaskBtPanelLeft:=16#1F;
ptrConfigPage^.wMaskBtPanelRight:=16#60;
ptrConfigPage^.wMaskFunctionPanel:=16#33;
(* Navigation panel restriction *)
ptrConfigPage^.wMaskTouchScreenNavPanel:=16#3F;
(* Active machine movement mask *)
ptrConfigPage^.wMaskActiveMachineBtPanelLeft:=16#0;
ptrConfigPage^.wMaskActiveMachineBtPanelRight:=16#0;
ptrConfigPage^.wMaskActiveMachineFunctionPanel:=16#0;
ptrConfigPage^.wMaskActiveMachineNavPanel:=16#3F;
(* Button edge action *)
ptrConfigPage^.aiRTrigActionPanelRight[1]:=10120;
ptrConfigPage^.aiRTrigActionPanelRight[2]:=10121;
ptrConfigPage^.aiRTrigActionPanelRight[3]:=0;
ptrConfigPage^.aiRTrigActionPanelRight[4]:=0;
ptrConfigPage^.aiRTrigActionPanelRight[5]:=0;
ptrConfigPage^.aiFTrigActionPanelRight[1]:=0;
ptrConfigPage^.aiFTrigActionPanelRight[2]:=0;
ptrConfigPage^.aiFTrigActionPanelRight[3]:=0;
ptrConfigPage^.aiFTrigActionPanelRight[4]:=0;
ptrConfigPage^.aiFTrigActionPanelRight[5]:=0;
ptrConfigPage^.aiDelayActionPanelRight[1]:=0;
ptrConfigPage^.aiDelayActionPanelRight[2]:=0;
ptrConfigPage^.aiDelayActionPanelRight[3]:=0;
ptrConfigPage^.aiDelayActionPanelRight[4]:=0;
ptrConfigPage^.aiDelayActionPanelRight[5]:=0;
ptrConfigPage^.aiRTrigActionFunctionPanel[1]:=206;
ptrConfigPage^.aiRTrigActionFunctionPanel[2]:=207;
ptrConfigPage^.aiRTrigActionFunctionPanel[3]:=0; (*Section 3&4 not used*)
ptrConfigPage^.aiRTrigActionFunctionPanel[4]:=0;
ptrConfigPage^.aiRTrigActionFunctionPanel[5]:=205;
ptrConfigPage^.aiRTrigActionFunctionPanel[6]:=1005;
ptrConfigPage^.aiRTrigActionFunctionPanel[7]:=0;
ptrConfigPage^.aiRTrigActionFunctionPanel[8]:=0;
ptrConfigPage^.aiRTrigActionFunctionPanel[9]:=0;
ptrConfigPage^.aiRTrigActionFunctionPanel[10]:=0;
ptrConfigPage^.aiRTrigActionFunctionPanel[11]:=0;
ptrConfigPage^.aiRTrigActionFunctionPanel[12]:=0;
ptrConfigPage^.aiFTrigActionTouchScreenNavPanel[1]:=10110;
ptrConfigPage^.aiFTrigActionTouchScreenNavPanel[2]:=10120;
ptrConfigPage^.aiFTrigActionTouchScreenNavPanel[3]:=10130;
ptrConfigPage^.aiFTrigActionTouchScreenNavPanel[4]:=10140;
ptrConfigPage^.aiFTrigActionTouchScreenNavPanel[5]:=10150;
ptrConfigPage^.aiFTrigActionTouchScreenNavPanel[6]:=10160;
ptrConfigPage^.xMaskBtStart:=FALSE;
ptrConfigPage^.xMaskBtStop:=TRUE;
END_ACTION
ACTION Page_130_Setup_Profile:
(* QVis page 130, Profile *)
iIndexPage:=130;
iPageNumber:=iPageNumber+1;
T_Visu.T_PageIndex[iIndexPage].iIndexConfigPage:=iPageNumber;
ptrConfigPage:=ADR(T_Visu.T_ConfigPage[T_Visu.T_PageIndex[iIndexPage].iIndexConfigPage]);
ptrConfigPage^.sName:='Profile';
ptrConfigPage^.wMaskBtPanelLeft:=16#1F;
ptrConfigPage^.wMaskBtPanelRight:=16#E0;
ptrConfigPage^.wMaskFunctionPanel:=16#0;
(* Navigation panel restriction *)
ptrConfigPage^.wMaskTouchScreenNavPanel:=16#3F;
(* Active machine movement mask *)
ptrConfigPage^.wMaskActiveMachineBtPanelLeft:=16#0;
ptrConfigPage^.wMaskActiveMachineBtPanelRight:=16#0;
ptrConfigPage^.wMaskActiveMachineFunctionPanel:=16#0;
ptrConfigPage^.wMaskActiveMachineNavPanel:=16#3F;
(* Button edge action *)
ptrConfigPage^.aiRTrigActionPanelRight[1]:=1002;
ptrConfigPage^.aiRTrigActionPanelRight[2]:=1003;
ptrConfigPage^.aiRTrigActionPanelRight[3]:=1004;
ptrConfigPage^.aiRTrigActionPanelRight[4]:=0;
ptrConfigPage^.aiRTrigActionPanelRight[5]:=0;
ptrConfigPage^.aiFTrigActionPanelRight[1]:=0;
ptrConfigPage^.aiFTrigActionPanelRight[2]:=0;
ptrConfigPage^.aiFTrigActionPanelRight[3]:=0;
ptrConfigPage^.aiFTrigActionPanelRight[4]:=0;
ptrConfigPage^.aiFTrigActionPanelRight[5]:=0;
ptrConfigPage^.aiDelayActionPanelRight[1]:=0;
ptrConfigPage^.aiDelayActionPanelRight[2]:=0;
ptrConfigPage^.aiDelayActionPanelRight[3]:=0;
ptrConfigPage^.aiDelayActionPanelRight[4]:=0;
ptrConfigPage^.aiDelayActionPanelRight[5]:=0;
ptrConfigPage^.aiRTrigActionFunctionPanel[1]:=0;
ptrConfigPage^.aiRTrigActionFunctionPanel[2]:=0;
ptrConfigPage^.aiRTrigActionFunctionPanel[3]:=0;
ptrConfigPage^.aiRTrigActionFunctionPanel[4]:=0;
ptrConfigPage^.aiRTrigActionFunctionPanel[5]:=0;
ptrConfigPage^.aiRTrigActionFunctionPanel[6]:=0;
ptrConfigPage^.aiRTrigActionFunctionPanel[7]:=0;
ptrConfigPage^.aiRTrigActionFunctionPanel[8]:=0;
ptrConfigPage^.aiRTrigActionFunctionPanel[9]:=0;
ptrConfigPage^.aiRTrigActionFunctionPanel[10]:=0;
ptrConfigPage^.aiRTrigActionFunctionPanel[11]:=0;
ptrConfigPage^.aiRTrigActionFunctionPanel[12]:=0;
ptrConfigPage^.aiFTrigActionTouchScreenNavPanel[1]:=10110;
ptrConfigPage^.aiFTrigActionTouchScreenNavPanel[2]:=10120;
ptrConfigPage^.aiFTrigActionTouchScreenNavPanel[3]:=10130;
ptrConfigPage^.aiFTrigActionTouchScreenNavPanel[4]:=10140;
ptrConfigPage^.aiFTrigActionTouchScreenNavPanel[5]:=10150;
ptrConfigPage^.aiFTrigActionTouchScreenNavPanel[6]:=10160;
ptrConfigPage^.xMaskBtStart:=FALSE;
ptrConfigPage^.xMaskBtStop:=TRUE;
END_ACTION
ACTION Page_140_Setup_Setup1:
(* QVis page 140, General Setup *)
iIndexPage:=140;
iPageNumber:=iPageNumber+1;
T_Visu.T_PageIndex[iIndexPage].iIndexConfigPage:=iPageNumber;
ptrConfigPage:=ADR(T_Visu.T_ConfigPage[T_Visu.T_PageIndex[iIndexPage].iIndexConfigPage]);
ptrConfigPage^.sName:='General Setup';
ptrConfigPage^.wMaskBtPanelLeft:=16#1F;
ptrConfigPage^.wMaskBtPanelRight:=16#60;
ptrConfigPage^.wMaskFunctionPanel:=16#0;
(* Navigation panel restriction *)
ptrConfigPage^.wMaskTouchScreenNavPanel:=16#3F;
(* Active machine movement mask *)
ptrConfigPage^.wMaskActiveMachineBtPanelLeft:=16#0;
ptrConfigPage^.wMaskActiveMachineBtPanelRight:=16#0;
ptrConfigPage^.wMaskActiveMachineFunctionPanel:=16#0;
ptrConfigPage^.wMaskActiveMachineNavPanel:=16#3F;
(* Button edge action *)
ptrConfigPage^.aiRTrigActionPanelRight[1]:=10140;
ptrConfigPage^.aiRTrigActionPanelRight[2]:=10141;
ptrConfigPage^.aiRTrigActionPanelRight[3]:=0;
ptrConfigPage^.aiRTrigActionPanelRight[4]:=0;
ptrConfigPage^.aiRTrigActionPanelRight[5]:=0;
ptrConfigPage^.aiFTrigActionPanelRight[1]:=0;
ptrConfigPage^.aiFTrigActionPanelRight[2]:=0;
ptrConfigPage^.aiFTrigActionPanelRight[3]:=0;
ptrConfigPage^.aiFTrigActionPanelRight[4]:=0;
ptrConfigPage^.aiFTrigActionPanelRight[5]:=0;
ptrConfigPage^.aiDelayActionPanelRight[1]:=0;
ptrConfigPage^.aiDelayActionPanelRight[2]:=0;
ptrConfigPage^.aiDelayActionPanelRight[3]:=0;
ptrConfigPage^.aiDelayActionPanelRight[4]:=0;
ptrConfigPage^.aiDelayActionPanelRight[5]:=0;
ptrConfigPage^.aiRTrigActionFunctionPanel[1]:=0;
ptrConfigPage^.aiRTrigActionFunctionPanel[2]:=0;
ptrConfigPage^.aiRTrigActionFunctionPanel[3]:=0;
ptrConfigPage^.aiRTrigActionFunctionPanel[4]:=0;
ptrConfigPage^.aiRTrigActionFunctionPanel[5]:=0;
ptrConfigPage^.aiRTrigActionFunctionPanel[6]:=0;
ptrConfigPage^.aiRTrigActionFunctionPanel[7]:=0;
ptrConfigPage^.aiRTrigActionFunctionPanel[8]:=0;
ptrConfigPage^.aiRTrigActionFunctionPanel[9]:=0;
ptrConfigPage^.aiRTrigActionFunctionPanel[10]:=0;
ptrConfigPage^.aiRTrigActionFunctionPanel[11]:=0;
ptrConfigPage^.aiRTrigActionFunctionPanel[12]:=0;
ptrConfigPage^.aiFTrigActionTouchScreenNavPanel[1]:=10110;
ptrConfigPage^.aiFTrigActionTouchScreenNavPanel[2]:=10120;
ptrConfigPage^.aiFTrigActionTouchScreenNavPanel[3]:=10130;
ptrConfigPage^.aiFTrigActionTouchScreenNavPanel[4]:=10140;
ptrConfigPage^.aiFTrigActionTouchScreenNavPanel[5]:=10150;
ptrConfigPage^.aiFTrigActionTouchScreenNavPanel[6]:=10160;
ptrConfigPage^.xMaskBtStart:=FALSE;
ptrConfigPage^.xMaskBtStop:=TRUE;
END_ACTION
ACTION Page_141_Setup_Setup2:
(*SOA 12.01.2023 {  *)
(* QVis page 141, Warm up *)
iIndexPage:=141;
iPageNumber:=iPageNumber+1;
T_Visu.T_PageIndex[iIndexPage].iIndexConfigPage:=iPageNumber;
ptrConfigPage:=ADR(T_Visu.T_ConfigPage[T_Visu.T_PageIndex[iIndexPage].iIndexConfigPage]);
ptrConfigPage^.sName:='Warm up';
ptrConfigPage^.wMaskBtPanelLeft:=16#1F;
ptrConfigPage^.wMaskBtPanelRight:=16#60;
ptrConfigPage^.wMaskFunctionPanel:=16#31;
(* Navigation panel restriction *)
ptrConfigPage^.wMaskTouchScreenNavPanel:=16#3F;
(* Active machine movement mask *)
ptrConfigPage^.wMaskActiveMachineBtPanelLeft:=16#0;
ptrConfigPage^.wMaskActiveMachineBtPanelRight:=16#0;
ptrConfigPage^.wMaskActiveMachineFunctionPanel:=16#0;
ptrConfigPage^.wMaskActiveMachineNavPanel:=16#3F;
(* Button edge action *)
ptrConfigPage^.aiRTrigActionPanelRight[1]:=10140;
ptrConfigPage^.aiRTrigActionPanelRight[2]:=10141;
ptrConfigPage^.aiRTrigActionPanelRight[3]:=0;
ptrConfigPage^.aiRTrigActionPanelRight[4]:=0;
ptrConfigPage^.aiRTrigActionPanelRight[5]:=0;
ptrConfigPage^.aiFTrigActionPanelRight[1]:=0;
ptrConfigPage^.aiFTrigActionPanelRight[2]:=0;
ptrConfigPage^.aiFTrigActionPanelRight[3]:=0;
ptrConfigPage^.aiFTrigActionPanelRight[4]:=0;
ptrConfigPage^.aiFTrigActionPanelRight[5]:=0;
ptrConfigPage^.aiDelayActionPanelRight[1]:=0;
ptrConfigPage^.aiDelayActionPanelRight[2]:=0;
ptrConfigPage^.aiDelayActionPanelRight[3]:=0;
ptrConfigPage^.aiDelayActionPanelRight[4]:=0;
ptrConfigPage^.aiDelayActionPanelRight[5]:=0;
ptrConfigPage^.aiRTrigActionFunctionPanel[1]:=173;
ptrConfigPage^.aiRTrigActionFunctionPanel[2]:=0;
ptrConfigPage^.aiRTrigActionFunctionPanel[3]:=0;
ptrConfigPage^.aiRTrigActionFunctionPanel[4]:=0;
ptrConfigPage^.aiRTrigActionFunctionPanel[5]:=175;
ptrConfigPage^.aiRTrigActionFunctionPanel[6]:= 1005; (*Vorher: 171*)
ptrConfigPage^.aiRTrigActionFunctionPanel[7]:=0;
ptrConfigPage^.aiRTrigActionFunctionPanel[8]:=0;
ptrConfigPage^.aiRTrigActionFunctionPanel[9]:=0;
ptrConfigPage^.aiRTrigActionFunctionPanel[10]:=0;
ptrConfigPage^.aiRTrigActionFunctionPanel[11]:=0;
ptrConfigPage^.aiRTrigActionFunctionPanel[12]:=0;
ptrConfigPage^.aiFTrigActionTouchScreenNavPanel[1]:=10110;
ptrConfigPage^.aiFTrigActionTouchScreenNavPanel[2]:=10120;
ptrConfigPage^.aiFTrigActionTouchScreenNavPanel[3]:=10130;
ptrConfigPage^.aiFTrigActionTouchScreenNavPanel[4]:=10140;
ptrConfigPage^.aiFTrigActionTouchScreenNavPanel[5]:=10150;
ptrConfigPage^.aiFTrigActionTouchScreenNavPanel[6]:=10160;
ptrConfigPage^.xMaskBtStart:=FALSE;
ptrConfigPage^.xMaskBtStop:=TRUE;
(*SOA 12.01.2023 }  *)
END_ACTION
ACTION Page_150_Setup_Config:
(* QVis page 150, Configuration *)
iIndexPage:=150;
iPageNumber:=iPageNumber+1;
T_Visu.T_PageIndex[iIndexPage].iIndexConfigPage:=iPageNumber;
ptrConfigPage:=ADR(T_Visu.T_ConfigPage[T_Visu.T_PageIndex[iIndexPage].iIndexConfigPage]);
ptrConfigPage^.sName:='Configuration';
ptrConfigPage^.wMaskBtPanelLeft:=16#1F;
ptrConfigPage^.wMaskBtPanelRight:=16#0;
ptrConfigPage^.wMaskFunctionPanel:=16#0;
(* Navigation panel restriction *)
ptrConfigPage^.wMaskTouchScreenNavPanel:=16#3F;
(* Active machine movement mask *)
ptrConfigPage^.wMaskActiveMachineBtPanelLeft:=16#0;
ptrConfigPage^.wMaskActiveMachineBtPanelRight:=16#0;
ptrConfigPage^.wMaskActiveMachineFunctionPanel:=16#0;
ptrConfigPage^.wMaskActiveMachineNavPanel:=16#3F;
(* Button edge action *)
ptrConfigPage^.aiRTrigActionPanelRight[1]:=0;
ptrConfigPage^.aiRTrigActionPanelRight[2]:=0;
ptrConfigPage^.aiRTrigActionPanelRight[3]:=0;
ptrConfigPage^.aiRTrigActionPanelRight[4]:=0;
ptrConfigPage^.aiRTrigActionPanelRight[5]:=0;
ptrConfigPage^.aiFTrigActionPanelRight[1]:=0;
ptrConfigPage^.aiFTrigActionPanelRight[2]:=0;
ptrConfigPage^.aiFTrigActionPanelRight[3]:=0;
ptrConfigPage^.aiFTrigActionPanelRight[4]:=0;
ptrConfigPage^.aiFTrigActionPanelRight[5]:=0;
ptrConfigPage^.aiDelayActionPanelRight[1]:=0;
ptrConfigPage^.aiDelayActionPanelRight[2]:=0;
ptrConfigPage^.aiDelayActionPanelRight[3]:=0;
ptrConfigPage^.aiDelayActionPanelRight[4]:=0;
ptrConfigPage^.aiDelayActionPanelRight[5]:=0;
ptrConfigPage^.aiRTrigActionFunctionPanel[1]:=0;
ptrConfigPage^.aiRTrigActionFunctionPanel[2]:=0;
ptrConfigPage^.aiRTrigActionFunctionPanel[3]:=0;
ptrConfigPage^.aiRTrigActionFunctionPanel[4]:=0;
ptrConfigPage^.aiRTrigActionFunctionPanel[5]:=0;
ptrConfigPage^.aiRTrigActionFunctionPanel[6]:=0;
ptrConfigPage^.aiRTrigActionFunctionPanel[7]:=0;
ptrConfigPage^.aiRTrigActionFunctionPanel[8]:=0;
ptrConfigPage^.aiRTrigActionFunctionPanel[9]:=0;
ptrConfigPage^.aiRTrigActionFunctionPanel[10]:=0;
ptrConfigPage^.aiRTrigActionFunctionPanel[11]:=0;
ptrConfigPage^.aiRTrigActionFunctionPanel[12]:=0;
ptrConfigPage^.aiFTrigActionTouchScreenNavPanel[1]:=10110;
ptrConfigPage^.aiFTrigActionTouchScreenNavPanel[2]:=10120;
ptrConfigPage^.aiFTrigActionTouchScreenNavPanel[3]:=10130;
ptrConfigPage^.aiFTrigActionTouchScreenNavPanel[4]:=10140;
ptrConfigPage^.aiFTrigActionTouchScreenNavPanel[5]:=10150;
ptrConfigPage^.aiFTrigActionTouchScreenNavPanel[6]:=10160;
ptrConfigPage^.xMaskBtStart:=FALSE;
ptrConfigPage^.xMaskBtStop:=TRUE;
END_ACTION
ACTION Page_160_Setup_ErrorList:
(* QVis page 160, Error List *)
iIndexPage:=160;
iPageNumber:=iPageNumber+1;
T_Visu.T_PageIndex[iIndexPage].iIndexConfigPage:=iPageNumber;
ptrConfigPage:=ADR(T_Visu.T_ConfigPage[T_Visu.T_PageIndex[iIndexPage].iIndexConfigPage]);
ptrConfigPage^.sName:='Error List';
ptrConfigPage^.wMaskBtPanelLeft:=16#1F;
ptrConfigPage^.wMaskBtPanelRight:=16#60;
ptrConfigPage^.wMaskFunctionPanel:=16#0;
(* Navigation panel restriction *)
ptrConfigPage^.wMaskTouchScreenNavPanel:=16#3F;
(* Active machine movement mask *)
ptrConfigPage^.wMaskActiveMachineBtPanelLeft:=16#0;
ptrConfigPage^.wMaskActiveMachineBtPanelRight:=16#60;
ptrConfigPage^.wMaskActiveMachineFunctionPanel:=16#0;
ptrConfigPage^.wMaskActiveMachineNavPanel:=16#3F;
(* Button edge action *)
ptrConfigPage^.aiRTrigActionPanelRight[1]:=99;
ptrConfigPage^.aiRTrigActionPanelRight[2]:=20;
ptrConfigPage^.aiRTrigActionPanelRight[3]:=0;
ptrConfigPage^.aiRTrigActionPanelRight[4]:=0;
ptrConfigPage^.aiRTrigActionPanelRight[5]:=0;
ptrConfigPage^.aiFTrigActionPanelRight[1]:=0;
ptrConfigPage^.aiFTrigActionPanelRight[2]:=0;
ptrConfigPage^.aiFTrigActionPanelRight[3]:=0;
ptrConfigPage^.aiFTrigActionPanelRight[4]:=0;
ptrConfigPage^.aiFTrigActionPanelRight[5]:=0;
ptrConfigPage^.aiDelayActionPanelRight[1]:=0;
ptrConfigPage^.aiDelayActionPanelRight[2]:=0;
ptrConfigPage^.aiDelayActionPanelRight[3]:=0;
ptrConfigPage^.aiDelayActionPanelRight[4]:=0;
ptrConfigPage^.aiDelayActionPanelRight[5]:=0;
ptrConfigPage^.aiRTrigActionFunctionPanel[1]:=0;
ptrConfigPage^.aiRTrigActionFunctionPanel[2]:=0;
ptrConfigPage^.aiRTrigActionFunctionPanel[3]:=0;
ptrConfigPage^.aiRTrigActionFunctionPanel[4]:=0;
ptrConfigPage^.aiRTrigActionFunctionPanel[5]:=0;
ptrConfigPage^.aiRTrigActionFunctionPanel[6]:=0;
ptrConfigPage^.aiRTrigActionFunctionPanel[7]:=0;
ptrConfigPage^.aiRTrigActionFunctionPanel[8]:=0;
ptrConfigPage^.aiRTrigActionFunctionPanel[9]:=0;
ptrConfigPage^.aiRTrigActionFunctionPanel[10]:=0;
ptrConfigPage^.aiRTrigActionFunctionPanel[11]:=0;
ptrConfigPage^.aiRTrigActionFunctionPanel[12]:=0;
ptrConfigPage^.aiFTrigActionTouchScreenNavPanel[1]:=10110;
ptrConfigPage^.aiFTrigActionTouchScreenNavPanel[2]:=10120;
ptrConfigPage^.aiFTrigActionTouchScreenNavPanel[3]:=10130;
ptrConfigPage^.aiFTrigActionTouchScreenNavPanel[4]:=10140;
ptrConfigPage^.aiFTrigActionTouchScreenNavPanel[5]:=10150;
ptrConfigPage^.aiFTrigActionTouchScreenNavPanel[6]:=10160;
ptrConfigPage^.xMaskBtStart:=FALSE;
ptrConfigPage^.xMaskBtStop:=TRUE;
END_ACTION
ACTION Page_170_Setup_Parameter:
(* QVis page 170, Parameter General *)
iIndexPage:=170;
iPageNumber:=iPageNumber+1;
T_Visu.T_PageIndex[iIndexPage].iIndexConfigPage:=iPageNumber;
ptrConfigPage:=ADR(T_Visu.T_ConfigPage[T_Visu.T_PageIndex[iIndexPage].iIndexConfigPage]);
ptrConfigPage^.sName:='Parameter General';
ptrConfigPage^.wMaskBtPanelLeft:=16#1F;
ptrConfigPage^.wMaskBtPanelRight:=16#200;
ptrConfigPage^.wMaskFunctionPanel:=16#0;
(* Navigation panel restriction *)
ptrConfigPage^.wMaskTouchScreenNavPanel:=16#3F;
(* Active machine movement mask *)
ptrConfigPage^.wMaskActiveMachineBtPanelLeft:=16#0;
ptrConfigPage^.wMaskActiveMachineBtPanelRight:=16#0;
ptrConfigPage^.wMaskActiveMachineFunctionPanel:=16#0;
ptrConfigPage^.wMaskActiveMachineNavPanel:=16#3F;
(* Button edge action *)
ptrConfigPage^.aiRTrigActionPanelRight[1]:=0;
ptrConfigPage^.aiRTrigActionPanelRight[2]:=0;
ptrConfigPage^.aiRTrigActionPanelRight[3]:=0;
ptrConfigPage^.aiRTrigActionPanelRight[4]:=0;
ptrConfigPage^.aiRTrigActionPanelRight[5]:=1006;
ptrConfigPage^.aiFTrigActionPanelRight[1]:=0;
ptrConfigPage^.aiFTrigActionPanelRight[2]:=0;
ptrConfigPage^.aiFTrigActionPanelRight[3]:=0;
ptrConfigPage^.aiFTrigActionPanelRight[4]:=0;
ptrConfigPage^.aiFTrigActionPanelRight[5]:=0;
ptrConfigPage^.aiDelayActionPanelRight[1]:=0;
ptrConfigPage^.aiDelayActionPanelRight[2]:=0;
ptrConfigPage^.aiDelayActionPanelRight[3]:=0;
ptrConfigPage^.aiDelayActionPanelRight[4]:=0;
ptrConfigPage^.aiDelayActionPanelRight[5]:=0;
ptrConfigPage^.aiRTrigActionFunctionPanel[1]:=0;
ptrConfigPage^.aiRTrigActionFunctionPanel[2]:=0;
ptrConfigPage^.aiRTrigActionFunctionPanel[3]:=0;
ptrConfigPage^.aiRTrigActionFunctionPanel[4]:=0;
ptrConfigPage^.aiRTrigActionFunctionPanel[5]:=0;
ptrConfigPage^.aiRTrigActionFunctionPanel[6]:=0;
ptrConfigPage^.aiRTrigActionFunctionPanel[7]:=0;
ptrConfigPage^.aiRTrigActionFunctionPanel[8]:=0;
ptrConfigPage^.aiRTrigActionFunctionPanel[9]:=0;
ptrConfigPage^.aiRTrigActionFunctionPanel[10]:=0;
ptrConfigPage^.aiRTrigActionFunctionPanel[11]:=0;
ptrConfigPage^.aiRTrigActionFunctionPanel[12]:=0;
ptrConfigPage^.aiFTrigActionTouchScreenNavPanel[1]:=10110;
ptrConfigPage^.aiFTrigActionTouchScreenNavPanel[2]:=10120;
ptrConfigPage^.aiFTrigActionTouchScreenNavPanel[3]:=10130;
ptrConfigPage^.aiFTrigActionTouchScreenNavPanel[4]:=10140;
ptrConfigPage^.aiFTrigActionTouchScreenNavPanel[5]:=10150;
ptrConfigPage^.aiFTrigActionTouchScreenNavPanel[6]:=10160;
ptrConfigPage^.xMaskBtStart:=FALSE;
ptrConfigPage^.xMaskBtStop:=TRUE;
END_ACTION
ACTION Page_210_WorkStation_Axis1:
(* QVis page 210, Teach-in Tool Rotation *)
iIndexPage:=210;
iPageNumber:=iPageNumber+1;
T_Visu.T_PageIndex[iIndexPage].iIndexConfigPage:=iPageNumber;
ptrConfigPage:=ADR(T_Visu.T_ConfigPage[T_Visu.T_PageIndex[iIndexPage].iIndexConfigPage]);
ptrConfigPage^.sName:='Teach-in Tool Rotation';
ptrConfigPage^.wMaskBtPanelLeft:=16#1F;
ptrConfigPage^.wMaskBtPanelRight:=16#1E0;
ptrConfigPage^.wMaskFunctionPanel:=16#F;
(* Navigation panel restriction *)
ptrConfigPage^.wMaskTouchScreenNavPanel:=16#27;
(* Active machine movement mask *)
ptrConfigPage^.wMaskActiveMachineBtPanelLeft:=16#0;
ptrConfigPage^.wMaskActiveMachineBtPanelRight:=16#0;
ptrConfigPage^.wMaskActiveMachineFunctionPanel:=16#0;
ptrConfigPage^.wMaskActiveMachineNavPanel:=16#27;
(* Button edge action *)
ptrConfigPage^.aiRTrigActionPanelRight[1]:=312;
ptrConfigPage^.aiRTrigActionPanelRight[2]:=310;
ptrConfigPage^.aiRTrigActionPanelRight[3]:=316;
ptrConfigPage^.aiRTrigActionPanelRight[4]:=314;
ptrConfigPage^.aiRTrigActionPanelRight[5]:=0;
ptrConfigPage^.aiFTrigActionPanelRight[1]:=0;
ptrConfigPage^.aiFTrigActionPanelRight[2]:=0;
ptrConfigPage^.aiFTrigActionPanelRight[3]:=301;
ptrConfigPage^.aiFTrigActionPanelRight[4]:=301;
ptrConfigPage^.aiFTrigActionPanelRight[5]:=0;
ptrConfigPage^.aiDelayActionPanelRight[1]:=0;
ptrConfigPage^.aiDelayActionPanelRight[2]:=0;
ptrConfigPage^.aiDelayActionPanelRight[3]:=0;
ptrConfigPage^.aiDelayActionPanelRight[4]:=0;
ptrConfigPage^.aiDelayActionPanelRight[5]:=0;
ptrConfigPage^.aiRTrigActionFunctionPanel[1]:=322;
ptrConfigPage^.aiRTrigActionFunctionPanel[2]:=323;
ptrConfigPage^.aiRTrigActionFunctionPanel[3]:=321;
ptrConfigPage^.aiRTrigActionFunctionPanel[4]:=320;
ptrConfigPage^.aiRTrigActionFunctionPanel[5]:=0;
ptrConfigPage^.aiRTrigActionFunctionPanel[6]:=0;
ptrConfigPage^.aiRTrigActionFunctionPanel[7]:=0;
ptrConfigPage^.aiRTrigActionFunctionPanel[8]:=0;
ptrConfigPage^.aiRTrigActionFunctionPanel[9]:=0;
ptrConfigPage^.aiRTrigActionFunctionPanel[10]:=0;
ptrConfigPage^.aiRTrigActionFunctionPanel[11]:=0;
ptrConfigPage^.aiRTrigActionFunctionPanel[12]:=0;
ptrConfigPage^.aiFTrigActionTouchScreenNavPanel[1]:=10210;
ptrConfigPage^.aiFTrigActionTouchScreenNavPanel[2]:=10220;
ptrConfigPage^.aiFTrigActionTouchScreenNavPanel[3]:=10230;
ptrConfigPage^.aiFTrigActionTouchScreenNavPanel[4]:=0;
ptrConfigPage^.aiFTrigActionTouchScreenNavPanel[5]:=0;
ptrConfigPage^.aiFTrigActionTouchScreenNavPanel[6]:=10260;
ptrConfigPage^.xMaskBtStart:=TRUE;
ptrConfigPage^.xMaskBtStop:=TRUE;
END_ACTION
ACTION Page_220_WorkStation_ToolTorque:
(* QVis page 220, Tool Torque *)
iIndexPage:=220;
iPageNumber:=iPageNumber+1;
T_Visu.T_PageIndex[iIndexPage].iIndexConfigPage:=iPageNumber;
ptrConfigPage:=ADR(T_Visu.T_ConfigPage[T_Visu.T_PageIndex[iIndexPage].iIndexConfigPage]);
ptrConfigPage^.sName:='Tool Torque';
ptrConfigPage^.wMaskBtPanelLeft:=16#1F;
ptrConfigPage^.wMaskBtPanelRight:=16#0;
ptrConfigPage^.wMaskFunctionPanel:=16#DF;
(* Navigation panel restriction *)
ptrConfigPage^.wMaskTouchScreenNavPanel:=16#27;
(* Active machine movement mask *)
ptrConfigPage^.wMaskActiveMachineBtPanelLeft:=16#0;
ptrConfigPage^.wMaskActiveMachineBtPanelRight:=16#0;
ptrConfigPage^.wMaskActiveMachineFunctionPanel:=16#DF;
ptrConfigPage^.wMaskActiveMachineNavPanel:=16#27;
(* Button edge action *)
ptrConfigPage^.aiRTrigActionPanelRight[1]:=0;
ptrConfigPage^.aiRTrigActionPanelRight[2]:=0;
ptrConfigPage^.aiRTrigActionPanelRight[3]:=0;
ptrConfigPage^.aiRTrigActionPanelRight[4]:=0;
ptrConfigPage^.aiRTrigActionPanelRight[5]:=0;
ptrConfigPage^.aiFTrigActionPanelRight[1]:=0;
ptrConfigPage^.aiFTrigActionPanelRight[2]:=0;
ptrConfigPage^.aiFTrigActionPanelRight[3]:=0;
ptrConfigPage^.aiFTrigActionPanelRight[4]:=0;
ptrConfigPage^.aiFTrigActionPanelRight[5]:=0;
ptrConfigPage^.aiDelayActionPanelRight[1]:=0;
ptrConfigPage^.aiDelayActionPanelRight[2]:=0;
ptrConfigPage^.aiDelayActionPanelRight[3]:=0;
ptrConfigPage^.aiDelayActionPanelRight[4]:=0;
ptrConfigPage^.aiDelayActionPanelRight[5]:=0;
ptrConfigPage^.aiRTrigActionFunctionPanel[1]:=502;
ptrConfigPage^.aiRTrigActionFunctionPanel[2]:=503;
ptrConfigPage^.aiRTrigActionFunctionPanel[3]:=501;
ptrConfigPage^.aiRTrigActionFunctionPanel[4]:=130;
ptrConfigPage^.aiRTrigActionFunctionPanel[5]:=131;
ptrConfigPage^.aiRTrigActionFunctionPanel[6]:=0;
ptrConfigPage^.aiRTrigActionFunctionPanel[7]:=504;
ptrConfigPage^.aiRTrigActionFunctionPanel[8]:=505;
ptrConfigPage^.aiRTrigActionFunctionPanel[9]:=0;
ptrConfigPage^.aiRTrigActionFunctionPanel[10]:=0;
ptrConfigPage^.aiRTrigActionFunctionPanel[11]:=0;
ptrConfigPage^.aiRTrigActionFunctionPanel[12]:=0;
ptrConfigPage^.aiFTrigActionTouchScreenNavPanel[1]:=10210;
ptrConfigPage^.aiFTrigActionTouchScreenNavPanel[2]:=10220;
ptrConfigPage^.aiFTrigActionTouchScreenNavPanel[3]:=10230;
ptrConfigPage^.aiFTrigActionTouchScreenNavPanel[4]:=0;
ptrConfigPage^.aiFTrigActionTouchScreenNavPanel[5]:=0;
ptrConfigPage^.aiFTrigActionTouchScreenNavPanel[6]:=10260;
ptrConfigPage^.xMaskBtStart:=TRUE;
ptrConfigPage^.xMaskBtStop:=TRUE;
END_ACTION
ACTION Page_230_WorkStation_ToolTension:
(* QVis page 230, Tool Tension *)
iIndexPage:=230;
iPageNumber:=iPageNumber+1;
T_Visu.T_PageIndex[iIndexPage].iIndexConfigPage:=iPageNumber;
ptrConfigPage:=ADR(T_Visu.T_ConfigPage[T_Visu.T_PageIndex[iIndexPage].iIndexConfigPage]);
ptrConfigPage^.sName:='Tool Tension';
ptrConfigPage^.wMaskBtPanelLeft:=16#1F;
ptrConfigPage^.wMaskBtPanelRight:=16#20;
ptrConfigPage^.wMaskFunctionPanel:=16#0;
(* Navigation panel restriction *)
ptrConfigPage^.wMaskTouchScreenNavPanel:=16#27;
(* Active machine movement mask *)
ptrConfigPage^.wMaskActiveMachineBtPanelLeft:=16#0;
ptrConfigPage^.wMaskActiveMachineBtPanelRight:=16#0;
ptrConfigPage^.wMaskActiveMachineFunctionPanel:=16#0;
ptrConfigPage^.wMaskActiveMachineNavPanel:=16#27;
(* Button edge action *)
ptrConfigPage^.aiRTrigActionPanelRight[1]:=501;
ptrConfigPage^.aiRTrigActionPanelRight[2]:=0;
ptrConfigPage^.aiRTrigActionPanelRight[3]:=0;
ptrConfigPage^.aiRTrigActionPanelRight[4]:=0;
ptrConfigPage^.aiRTrigActionPanelRight[5]:=0;
ptrConfigPage^.aiFTrigActionPanelRight[1]:=0;
ptrConfigPage^.aiFTrigActionPanelRight[2]:=0;
ptrConfigPage^.aiFTrigActionPanelRight[3]:=0;
ptrConfigPage^.aiFTrigActionPanelRight[4]:=0;
ptrConfigPage^.aiFTrigActionPanelRight[5]:=0;
ptrConfigPage^.aiDelayActionPanelRight[1]:=0;
ptrConfigPage^.aiDelayActionPanelRight[2]:=0;
ptrConfigPage^.aiDelayActionPanelRight[3]:=0;
ptrConfigPage^.aiDelayActionPanelRight[4]:=0;
ptrConfigPage^.aiDelayActionPanelRight[5]:=0;
ptrConfigPage^.aiRTrigActionFunctionPanel[1]:=0;
ptrConfigPage^.aiRTrigActionFunctionPanel[2]:=0;
ptrConfigPage^.aiRTrigActionFunctionPanel[3]:=0;
ptrConfigPage^.aiRTrigActionFunctionPanel[4]:=0;
ptrConfigPage^.aiRTrigActionFunctionPanel[5]:=0;
ptrConfigPage^.aiRTrigActionFunctionPanel[6]:=0;
ptrConfigPage^.aiRTrigActionFunctionPanel[7]:=0;
ptrConfigPage^.aiRTrigActionFunctionPanel[8]:=0;
ptrConfigPage^.aiRTrigActionFunctionPanel[9]:=0;
ptrConfigPage^.aiRTrigActionFunctionPanel[10]:=0;
ptrConfigPage^.aiRTrigActionFunctionPanel[11]:=0;
ptrConfigPage^.aiRTrigActionFunctionPanel[12]:=0;
ptrConfigPage^.aiFTrigActionTouchScreenNavPanel[1]:=10210;
ptrConfigPage^.aiFTrigActionTouchScreenNavPanel[2]:=10220;
ptrConfigPage^.aiFTrigActionTouchScreenNavPanel[3]:=10230;
ptrConfigPage^.aiFTrigActionTouchScreenNavPanel[4]:=0;
ptrConfigPage^.aiFTrigActionTouchScreenNavPanel[5]:=0;
ptrConfigPage^.aiFTrigActionTouchScreenNavPanel[6]:=10260;
ptrConfigPage^.xMaskBtStart:=FALSE;
ptrConfigPage^.xMaskBtStop:=TRUE;
END_ACTION
ACTION Page_260_WorkStation_ErrorList:
(* QVis page 260, Error List *)
iIndexPage:=260;
iPageNumber:=iPageNumber+1;
T_Visu.T_PageIndex[iIndexPage].iIndexConfigPage:=iPageNumber;
ptrConfigPage:=ADR(T_Visu.T_ConfigPage[T_Visu.T_PageIndex[iIndexPage].iIndexConfigPage]);
ptrConfigPage^.sName:='Error List';
ptrConfigPage^.wMaskBtPanelLeft:=16#1F;
ptrConfigPage^.wMaskBtPanelRight:=16#60;
ptrConfigPage^.wMaskFunctionPanel:=16#0;
(* Navigation panel restriction *)
ptrConfigPage^.wMaskTouchScreenNavPanel:=16#27;
(* Active machine movement mask *)
ptrConfigPage^.wMaskActiveMachineBtPanelLeft:=16#0;
ptrConfigPage^.wMaskActiveMachineBtPanelRight:=16#60;
ptrConfigPage^.wMaskActiveMachineFunctionPanel:=16#0;
ptrConfigPage^.wMaskActiveMachineNavPanel:=16#27;
(* Button edge action *)
ptrConfigPage^.aiRTrigActionPanelRight[1]:=99;
ptrConfigPage^.aiRTrigActionPanelRight[2]:=20;
ptrConfigPage^.aiRTrigActionPanelRight[3]:=0;
ptrConfigPage^.aiRTrigActionPanelRight[4]:=0;
ptrConfigPage^.aiRTrigActionPanelRight[5]:=0;
ptrConfigPage^.aiFTrigActionPanelRight[1]:=0;
ptrConfigPage^.aiFTrigActionPanelRight[2]:=0;
ptrConfigPage^.aiFTrigActionPanelRight[3]:=0;
ptrConfigPage^.aiFTrigActionPanelRight[4]:=0;
ptrConfigPage^.aiFTrigActionPanelRight[5]:=0;
ptrConfigPage^.aiDelayActionPanelRight[1]:=0;
ptrConfigPage^.aiDelayActionPanelRight[2]:=0;
ptrConfigPage^.aiDelayActionPanelRight[3]:=0;
ptrConfigPage^.aiDelayActionPanelRight[4]:=0;
ptrConfigPage^.aiDelayActionPanelRight[5]:=0;
ptrConfigPage^.aiRTrigActionFunctionPanel[1]:=0;
ptrConfigPage^.aiRTrigActionFunctionPanel[2]:=0;
ptrConfigPage^.aiRTrigActionFunctionPanel[3]:=0;
ptrConfigPage^.aiRTrigActionFunctionPanel[4]:=0;
ptrConfigPage^.aiRTrigActionFunctionPanel[5]:=0;
ptrConfigPage^.aiRTrigActionFunctionPanel[6]:=0;
ptrConfigPage^.aiRTrigActionFunctionPanel[7]:=0;
ptrConfigPage^.aiRTrigActionFunctionPanel[8]:=0;
ptrConfigPage^.aiRTrigActionFunctionPanel[9]:=0;
ptrConfigPage^.aiRTrigActionFunctionPanel[10]:=0;
ptrConfigPage^.aiRTrigActionFunctionPanel[11]:=0;
ptrConfigPage^.aiRTrigActionFunctionPanel[12]:=0;
ptrConfigPage^.aiFTrigActionTouchScreenNavPanel[1]:=10210;
ptrConfigPage^.aiFTrigActionTouchScreenNavPanel[2]:=10220;
ptrConfigPage^.aiFTrigActionTouchScreenNavPanel[3]:=10230;
ptrConfigPage^.aiFTrigActionTouchScreenNavPanel[4]:=0;
ptrConfigPage^.aiFTrigActionTouchScreenNavPanel[5]:=0;
ptrConfigPage^.aiFTrigActionTouchScreenNavPanel[6]:=10260;
ptrConfigPage^.xMaskBtStart:=FALSE;
ptrConfigPage^.xMaskBtStop:=TRUE;
END_ACTION
ACTION Page_270_WorkStation_Parameter1:
(* QVis page 270, Parameter Tool Rotation *)
iIndexPage:=270;
iPageNumber:=iPageNumber+1;
T_Visu.T_PageIndex[iIndexPage].iIndexConfigPage:=iPageNumber;
ptrConfigPage:=ADR(T_Visu.T_ConfigPage[T_Visu.T_PageIndex[iIndexPage].iIndexConfigPage]);
ptrConfigPage^.sName:='Parameter Tool Rotation';
ptrConfigPage^.wMaskBtPanelLeft:=16#1F;
ptrConfigPage^.wMaskBtPanelRight:=16#200;
ptrConfigPage^.wMaskFunctionPanel:=16#0;
(* Navigation panel restriction *)
ptrConfigPage^.wMaskTouchScreenNavPanel:=16#27;
(* Active machine movement mask *)
ptrConfigPage^.wMaskActiveMachineBtPanelLeft:=16#0;
ptrConfigPage^.wMaskActiveMachineBtPanelRight:=16#0;
ptrConfigPage^.wMaskActiveMachineFunctionPanel:=16#0;
ptrConfigPage^.wMaskActiveMachineNavPanel:=16#27;
(* Button edge action *)
ptrConfigPage^.aiRTrigActionPanelRight[1]:=0;
ptrConfigPage^.aiRTrigActionPanelRight[2]:=0;
ptrConfigPage^.aiRTrigActionPanelRight[3]:=0;
ptrConfigPage^.aiRTrigActionPanelRight[4]:=0;
ptrConfigPage^.aiRTrigActionPanelRight[5]:=1006;
ptrConfigPage^.aiFTrigActionPanelRight[1]:=0;
ptrConfigPage^.aiFTrigActionPanelRight[2]:=0;
ptrConfigPage^.aiFTrigActionPanelRight[3]:=0;
ptrConfigPage^.aiFTrigActionPanelRight[4]:=0;
ptrConfigPage^.aiFTrigActionPanelRight[5]:=0;
ptrConfigPage^.aiDelayActionPanelRight[1]:=0;
ptrConfigPage^.aiDelayActionPanelRight[2]:=0;
ptrConfigPage^.aiDelayActionPanelRight[3]:=0;
ptrConfigPage^.aiDelayActionPanelRight[4]:=0;
ptrConfigPage^.aiDelayActionPanelRight[5]:=0;
ptrConfigPage^.aiRTrigActionFunctionPanel[1]:=0;
ptrConfigPage^.aiRTrigActionFunctionPanel[2]:=0;
ptrConfigPage^.aiRTrigActionFunctionPanel[3]:=0;
ptrConfigPage^.aiRTrigActionFunctionPanel[4]:=0;
ptrConfigPage^.aiRTrigActionFunctionPanel[5]:=0;
ptrConfigPage^.aiRTrigActionFunctionPanel[6]:=0;
ptrConfigPage^.aiRTrigActionFunctionPanel[7]:=0;
ptrConfigPage^.aiRTrigActionFunctionPanel[8]:=0;
ptrConfigPage^.aiRTrigActionFunctionPanel[9]:=0;
ptrConfigPage^.aiRTrigActionFunctionPanel[10]:=0;
ptrConfigPage^.aiRTrigActionFunctionPanel[11]:=0;
ptrConfigPage^.aiRTrigActionFunctionPanel[12]:=0;
ptrConfigPage^.aiFTrigActionTouchScreenNavPanel[1]:=10210;
ptrConfigPage^.aiFTrigActionTouchScreenNavPanel[2]:=10220;
ptrConfigPage^.aiFTrigActionTouchScreenNavPanel[3]:=10230;
ptrConfigPage^.aiFTrigActionTouchScreenNavPanel[4]:=0;
ptrConfigPage^.aiFTrigActionTouchScreenNavPanel[5]:=0;
ptrConfigPage^.aiFTrigActionTouchScreenNavPanel[6]:=10260;
ptrConfigPage^.xMaskBtStart:=FALSE;
ptrConfigPage^.xMaskBtStop:=TRUE;
END_ACTION
ACTION Page_310_WorkStation_Axis2:
(* QVis page 310, Teach-in Wire Feeder *)
iIndexPage:=310;
iPageNumber:=iPageNumber+1;
T_Visu.T_PageIndex[iIndexPage].iIndexConfigPage:=iPageNumber;
ptrConfigPage:=ADR(T_Visu.T_ConfigPage[T_Visu.T_PageIndex[iIndexPage].iIndexConfigPage]);
ptrConfigPage^.sName:='Teach-in Wire Feeder';
ptrConfigPage^.wMaskBtPanelLeft:=16#1F;
ptrConfigPage^.wMaskBtPanelRight:=16#1E0;
ptrConfigPage^.wMaskFunctionPanel:=16#3F;
(* Navigation panel restriction *)
ptrConfigPage^.wMaskTouchScreenNavPanel:=16#27;
(* Active machine movement mask *)
ptrConfigPage^.wMaskActiveMachineBtPanelLeft:=16#0;
ptrConfigPage^.wMaskActiveMachineBtPanelRight:=16#0;
ptrConfigPage^.wMaskActiveMachineFunctionPanel:=16#0;
ptrConfigPage^.wMaskActiveMachineNavPanel:=16#27;
(* Button edge action *)
ptrConfigPage^.aiRTrigActionPanelRight[1]:=312;
ptrConfigPage^.aiRTrigActionPanelRight[2]:=310;
ptrConfigPage^.aiRTrigActionPanelRight[3]:=316;
ptrConfigPage^.aiRTrigActionPanelRight[4]:=314;
ptrConfigPage^.aiRTrigActionPanelRight[5]:=0;
ptrConfigPage^.aiFTrigActionPanelRight[1]:=0;
ptrConfigPage^.aiFTrigActionPanelRight[2]:=0;
ptrConfigPage^.aiFTrigActionPanelRight[3]:=301;
ptrConfigPage^.aiFTrigActionPanelRight[4]:=301;
ptrConfigPage^.aiFTrigActionPanelRight[5]:=0;
ptrConfigPage^.aiDelayActionPanelRight[1]:=0;
ptrConfigPage^.aiDelayActionPanelRight[2]:=0;
ptrConfigPage^.aiDelayActionPanelRight[3]:=0;
ptrConfigPage^.aiDelayActionPanelRight[4]:=0;
ptrConfigPage^.aiDelayActionPanelRight[5]:=0;
ptrConfigPage^.aiRTrigActionFunctionPanel[1]:=322;
ptrConfigPage^.aiRTrigActionFunctionPanel[2]:=323;
ptrConfigPage^.aiRTrigActionFunctionPanel[3]:=324;
ptrConfigPage^.aiRTrigActionFunctionPanel[4]:=320;
ptrConfigPage^.aiRTrigActionFunctionPanel[5]:=501;
ptrConfigPage^.aiRTrigActionFunctionPanel[6]:=325;
ptrConfigPage^.aiRTrigActionFunctionPanel[7]:=0;
ptrConfigPage^.aiRTrigActionFunctionPanel[8]:=0;
ptrConfigPage^.aiRTrigActionFunctionPanel[9]:=0;
ptrConfigPage^.aiRTrigActionFunctionPanel[10]:=0;
ptrConfigPage^.aiRTrigActionFunctionPanel[11]:=0;
ptrConfigPage^.aiRTrigActionFunctionPanel[12]:=0;
ptrConfigPage^.aiFTrigActionTouchScreenNavPanel[1]:=10310;
ptrConfigPage^.aiFTrigActionTouchScreenNavPanel[2]:=10320;
ptrConfigPage^.aiFTrigActionTouchScreenNavPanel[3]:=10330;
ptrConfigPage^.aiFTrigActionTouchScreenNavPanel[4]:=0;
ptrConfigPage^.aiFTrigActionTouchScreenNavPanel[5]:=0;
ptrConfigPage^.aiFTrigActionTouchScreenNavPanel[6]:=10360;
ptrConfigPage^.xMaskBtStart:=TRUE;
ptrConfigPage^.xMaskBtStop:=TRUE;
END_ACTION
ACTION Page_320_WorkStation_SettingUp:
(* QVis page 320, Setting-up *)
iIndexPage:=320;
iPageNumber:=iPageNumber+1;
T_Visu.T_PageIndex[iIndexPage].iIndexConfigPage:=iPageNumber;
ptrConfigPage:=ADR(T_Visu.T_ConfigPage[T_Visu.T_PageIndex[iIndexPage].iIndexConfigPage]);
ptrConfigPage^.sName:='Setting-up';
ptrConfigPage^.wMaskBtPanelLeft:=16#1F;
ptrConfigPage^.wMaskBtPanelRight:=16#60;
ptrConfigPage^.wMaskFunctionPanel:=16#F;
(* Navigation panel restriction *)
ptrConfigPage^.wMaskTouchScreenNavPanel:=16#27;
(* Active machine movement mask *)
ptrConfigPage^.wMaskActiveMachineBtPanelLeft:=16#0;
ptrConfigPage^.wMaskActiveMachineBtPanelRight:=16#0;
ptrConfigPage^.wMaskActiveMachineFunctionPanel:=16#0;
ptrConfigPage^.wMaskActiveMachineNavPanel:=16#27;
(* Button edge action *)
ptrConfigPage^.aiRTrigActionPanelRight[1]:=312;
ptrConfigPage^.aiRTrigActionPanelRight[2]:=310;
ptrConfigPage^.aiRTrigActionPanelRight[3]:=0;
ptrConfigPage^.aiRTrigActionPanelRight[4]:=0;
ptrConfigPage^.aiRTrigActionPanelRight[5]:=0;
ptrConfigPage^.aiFTrigActionPanelRight[1]:=301;
ptrConfigPage^.aiFTrigActionPanelRight[2]:=301;
ptrConfigPage^.aiFTrigActionPanelRight[3]:=0;
ptrConfigPage^.aiFTrigActionPanelRight[4]:=0;
ptrConfigPage^.aiFTrigActionPanelRight[5]:=0;
ptrConfigPage^.aiDelayActionPanelRight[1]:=316;
ptrConfigPage^.aiDelayActionPanelRight[2]:=314;
ptrConfigPage^.aiDelayActionPanelRight[3]:=0;
ptrConfigPage^.aiDelayActionPanelRight[4]:=0;
ptrConfigPage^.aiDelayActionPanelRight[5]:=0;
ptrConfigPage^.aiRTrigActionFunctionPanel[1]:=322;
ptrConfigPage^.aiRTrigActionFunctionPanel[2]:=323;
ptrConfigPage^.aiRTrigActionFunctionPanel[3]:=326;
ptrConfigPage^.aiRTrigActionFunctionPanel[4]:=320;
ptrConfigPage^.aiRTrigActionFunctionPanel[5]:=0;
ptrConfigPage^.aiRTrigActionFunctionPanel[6]:=0;
ptrConfigPage^.aiRTrigActionFunctionPanel[7]:=0;
ptrConfigPage^.aiRTrigActionFunctionPanel[8]:=0;
ptrConfigPage^.aiRTrigActionFunctionPanel[9]:=0;
ptrConfigPage^.aiRTrigActionFunctionPanel[10]:=0;
ptrConfigPage^.aiRTrigActionFunctionPanel[11]:=0;
ptrConfigPage^.aiRTrigActionFunctionPanel[12]:=0;
ptrConfigPage^.aiFTrigActionTouchScreenNavPanel[1]:=10310;
ptrConfigPage^.aiFTrigActionTouchScreenNavPanel[2]:=10320;
ptrConfigPage^.aiFTrigActionTouchScreenNavPanel[3]:=10330;
ptrConfigPage^.aiFTrigActionTouchScreenNavPanel[4]:=0;
ptrConfigPage^.aiFTrigActionTouchScreenNavPanel[5]:=0;
ptrConfigPage^.aiFTrigActionTouchScreenNavPanel[6]:=10360;
ptrConfigPage^.xMaskBtStart:=FALSE;
ptrConfigPage^.xMaskBtStop:=TRUE;
END_ACTION
ACTION Page_330_WorkStation_Reference:
(* QVis page 330, ReferenceMaxToolLength *)
iIndexPage:=330;
iPageNumber:=iPageNumber+1;
T_Visu.T_PageIndex[iIndexPage].iIndexConfigPage:=iPageNumber;
ptrConfigPage:=ADR(T_Visu.T_ConfigPage[T_Visu.T_PageIndex[iIndexPage].iIndexConfigPage]);
ptrConfigPage^.sName:='Reference max ToolLength';
ptrConfigPage^.wMaskBtPanelLeft:=16#1F;
ptrConfigPage^.wMaskBtPanelRight:=16#1E0;
ptrConfigPage^.wMaskFunctionPanel:=16#1B;
(* Navigation panel restriction *)
ptrConfigPage^.wMaskTouchScreenNavPanel:=16#27;
(* Active machine movement mask *)
ptrConfigPage^.wMaskActiveMachineBtPanelLeft:=16#0;
ptrConfigPage^.wMaskActiveMachineBtPanelRight:=16#0;
ptrConfigPage^.wMaskActiveMachineFunctionPanel:=16#0;
ptrConfigPage^.wMaskActiveMachineNavPanel:=16#27;
(* Button edge action *)
ptrConfigPage^.aiRTrigActionPanelRight[1]:=312;
ptrConfigPage^.aiRTrigActionPanelRight[2]:=310;
ptrConfigPage^.aiRTrigActionPanelRight[3]:=316;
ptrConfigPage^.aiRTrigActionPanelRight[4]:=314;
ptrConfigPage^.aiRTrigActionPanelRight[5]:=0;
ptrConfigPage^.aiFTrigActionPanelRight[1]:=0;
ptrConfigPage^.aiFTrigActionPanelRight[2]:=0;
ptrConfigPage^.aiFTrigActionPanelRight[3]:=301;
ptrConfigPage^.aiFTrigActionPanelRight[4]:=301;
ptrConfigPage^.aiFTrigActionPanelRight[5]:=0;
ptrConfigPage^.aiDelayActionPanelRight[1]:=0;
ptrConfigPage^.aiDelayActionPanelRight[2]:=0;
ptrConfigPage^.aiDelayActionPanelRight[3]:=0;
ptrConfigPage^.aiDelayActionPanelRight[4]:=0;
ptrConfigPage^.aiDelayActionPanelRight[5]:=0;
ptrConfigPage^.aiRTrigActionFunctionPanel[1]:=322;
ptrConfigPage^.aiRTrigActionFunctionPanel[2]:=323;
ptrConfigPage^.aiRTrigActionFunctionPanel[3]:=0;
ptrConfigPage^.aiRTrigActionFunctionPanel[4]:=320;
ptrConfigPage^.aiRTrigActionFunctionPanel[5]:=501;
ptrConfigPage^.aiRTrigActionFunctionPanel[6]:=0;
ptrConfigPage^.aiRTrigActionFunctionPanel[7]:=0;
ptrConfigPage^.aiRTrigActionFunctionPanel[8]:=0;
ptrConfigPage^.aiRTrigActionFunctionPanel[9]:=0;
ptrConfigPage^.aiRTrigActionFunctionPanel[10]:=0;
ptrConfigPage^.aiRTrigActionFunctionPanel[11]:=0;
ptrConfigPage^.aiRTrigActionFunctionPanel[12]:=0;
ptrConfigPage^.aiFTrigActionTouchScreenNavPanel[1]:=10310;
ptrConfigPage^.aiFTrigActionTouchScreenNavPanel[2]:=10320;
ptrConfigPage^.aiFTrigActionTouchScreenNavPanel[3]:=10330;
ptrConfigPage^.aiFTrigActionTouchScreenNavPanel[4]:=0;
ptrConfigPage^.aiFTrigActionTouchScreenNavPanel[5]:=0;
ptrConfigPage^.aiFTrigActionTouchScreenNavPanel[6]:=10360;
ptrConfigPage^.xMaskBtStart:=TRUE;
ptrConfigPage^.xMaskBtStop:=TRUE;
END_ACTION
ACTION Page_360_WorkStation_ErrorList:
(* QVis page 360, Error List *)
iIndexPage:=360;
iPageNumber:=iPageNumber+1;
T_Visu.T_PageIndex[iIndexPage].iIndexConfigPage:=iPageNumber;
ptrConfigPage:=ADR(T_Visu.T_ConfigPage[T_Visu.T_PageIndex[iIndexPage].iIndexConfigPage]);
ptrConfigPage^.sName:='Error List';
ptrConfigPage^.wMaskBtPanelLeft:=16#1F;
ptrConfigPage^.wMaskBtPanelRight:=16#60;
ptrConfigPage^.wMaskFunctionPanel:=16#0;
(* Navigation panel restriction *)
ptrConfigPage^.wMaskTouchScreenNavPanel:=16#27;
(* Active machine movement mask *)
ptrConfigPage^.wMaskActiveMachineBtPanelLeft:=16#0;
ptrConfigPage^.wMaskActiveMachineBtPanelRight:=16#60;
ptrConfigPage^.wMaskActiveMachineFunctionPanel:=16#0;
ptrConfigPage^.wMaskActiveMachineNavPanel:=16#27;
(* Button edge action *)
ptrConfigPage^.aiRTrigActionPanelRight[1]:=99;
ptrConfigPage^.aiRTrigActionPanelRight[2]:=20;
ptrConfigPage^.aiRTrigActionPanelRight[3]:=0;
ptrConfigPage^.aiRTrigActionPanelRight[4]:=0;
ptrConfigPage^.aiRTrigActionPanelRight[5]:=0;
ptrConfigPage^.aiFTrigActionPanelRight[1]:=0;
ptrConfigPage^.aiFTrigActionPanelRight[2]:=0;
ptrConfigPage^.aiFTrigActionPanelRight[3]:=0;
ptrConfigPage^.aiFTrigActionPanelRight[4]:=0;
ptrConfigPage^.aiFTrigActionPanelRight[5]:=0;
ptrConfigPage^.aiDelayActionPanelRight[1]:=0;
ptrConfigPage^.aiDelayActionPanelRight[2]:=0;
ptrConfigPage^.aiDelayActionPanelRight[3]:=0;
ptrConfigPage^.aiDelayActionPanelRight[4]:=0;
ptrConfigPage^.aiDelayActionPanelRight[5]:=0;
ptrConfigPage^.aiRTrigActionFunctionPanel[1]:=0;
ptrConfigPage^.aiRTrigActionFunctionPanel[2]:=0;
ptrConfigPage^.aiRTrigActionFunctionPanel[3]:=0;
ptrConfigPage^.aiRTrigActionFunctionPanel[4]:=0;
ptrConfigPage^.aiRTrigActionFunctionPanel[5]:=0;
ptrConfigPage^.aiRTrigActionFunctionPanel[6]:=0;
ptrConfigPage^.aiRTrigActionFunctionPanel[7]:=0;
ptrConfigPage^.aiRTrigActionFunctionPanel[8]:=0;
ptrConfigPage^.aiRTrigActionFunctionPanel[9]:=0;
ptrConfigPage^.aiRTrigActionFunctionPanel[10]:=0;
ptrConfigPage^.aiRTrigActionFunctionPanel[11]:=0;
ptrConfigPage^.aiRTrigActionFunctionPanel[12]:=0;
ptrConfigPage^.aiFTrigActionTouchScreenNavPanel[1]:=10310;
ptrConfigPage^.aiFTrigActionTouchScreenNavPanel[2]:=10320;
ptrConfigPage^.aiFTrigActionTouchScreenNavPanel[3]:=10330;
ptrConfigPage^.aiFTrigActionTouchScreenNavPanel[4]:=0;
ptrConfigPage^.aiFTrigActionTouchScreenNavPanel[5]:=0;
ptrConfigPage^.aiFTrigActionTouchScreenNavPanel[6]:=10360;
ptrConfigPage^.xMaskBtStart:=FALSE;
ptrConfigPage^.xMaskBtStop:=TRUE;
END_ACTION
ACTION Page_370_WorkStation_Parameter2:
(* QVis page 370, Parameter Wire Feeder *)
iIndexPage:=370;
iPageNumber:=iPageNumber+1;
T_Visu.T_PageIndex[iIndexPage].iIndexConfigPage:=iPageNumber;
ptrConfigPage:=ADR(T_Visu.T_ConfigPage[T_Visu.T_PageIndex[iIndexPage].iIndexConfigPage]);
ptrConfigPage^.sName:='Parameter Wire Feeder';
ptrConfigPage^.wMaskBtPanelLeft:=16#1F;
ptrConfigPage^.wMaskBtPanelRight:=16#200;
ptrConfigPage^.wMaskFunctionPanel:=16#0;
(* Navigation panel restriction *)
ptrConfigPage^.wMaskTouchScreenNavPanel:=16#27;
(* Active machine movement mask *)
ptrConfigPage^.wMaskActiveMachineBtPanelLeft:=16#0;
ptrConfigPage^.wMaskActiveMachineBtPanelRight:=16#0;
ptrConfigPage^.wMaskActiveMachineFunctionPanel:=16#0;
ptrConfigPage^.wMaskActiveMachineNavPanel:=16#27;
(* Button edge action *)
ptrConfigPage^.aiRTrigActionPanelRight[1]:=0;
ptrConfigPage^.aiRTrigActionPanelRight[2]:=0;
ptrConfigPage^.aiRTrigActionPanelRight[3]:=0;
ptrConfigPage^.aiRTrigActionPanelRight[4]:=0;
ptrConfigPage^.aiRTrigActionPanelRight[5]:=1006;
ptrConfigPage^.aiFTrigActionPanelRight[1]:=0;
ptrConfigPage^.aiFTrigActionPanelRight[2]:=0;
ptrConfigPage^.aiFTrigActionPanelRight[3]:=0;
ptrConfigPage^.aiFTrigActionPanelRight[4]:=0;
ptrConfigPage^.aiFTrigActionPanelRight[5]:=0;
ptrConfigPage^.aiDelayActionPanelRight[1]:=0;
ptrConfigPage^.aiDelayActionPanelRight[2]:=0;
ptrConfigPage^.aiDelayActionPanelRight[3]:=0;
ptrConfigPage^.aiDelayActionPanelRight[4]:=0;
ptrConfigPage^.aiDelayActionPanelRight[5]:=0;
ptrConfigPage^.aiRTrigActionFunctionPanel[1]:=0;
ptrConfigPage^.aiRTrigActionFunctionPanel[2]:=0;
ptrConfigPage^.aiRTrigActionFunctionPanel[3]:=0;
ptrConfigPage^.aiRTrigActionFunctionPanel[4]:=0;
ptrConfigPage^.aiRTrigActionFunctionPanel[5]:=0;
ptrConfigPage^.aiRTrigActionFunctionPanel[6]:=0;
ptrConfigPage^.aiRTrigActionFunctionPanel[7]:=0;
ptrConfigPage^.aiRTrigActionFunctionPanel[8]:=0;
ptrConfigPage^.aiRTrigActionFunctionPanel[9]:=0;
ptrConfigPage^.aiRTrigActionFunctionPanel[10]:=0;
ptrConfigPage^.aiRTrigActionFunctionPanel[11]:=0;
ptrConfigPage^.aiRTrigActionFunctionPanel[12]:=0;
ptrConfigPage^.aiFTrigActionTouchScreenNavPanel[1]:=10310;
ptrConfigPage^.aiFTrigActionTouchScreenNavPanel[2]:=10320;
ptrConfigPage^.aiFTrigActionTouchScreenNavPanel[3]:=10330;
ptrConfigPage^.aiFTrigActionTouchScreenNavPanel[4]:=0;
ptrConfigPage^.aiFTrigActionTouchScreenNavPanel[5]:=0;
ptrConfigPage^.aiFTrigActionTouchScreenNavPanel[6]:=10360;
ptrConfigPage^.xMaskBtStart:=FALSE;
ptrConfigPage^.xMaskBtStop:=TRUE;
END_ACTION
ACTION Page_410_WorkStation_Axis3:
(* QVis page 410, Teach-in Grind Axis *)
iIndexPage:=410;
iPageNumber:=iPageNumber+1;
T_Visu.T_PageIndex[iIndexPage].iIndexConfigPage:=iPageNumber;
ptrConfigPage:=ADR(T_Visu.T_ConfigPage[T_Visu.T_PageIndex[iIndexPage].iIndexConfigPage]);
ptrConfigPage^.sName:='Teach-in Grind Axis';
ptrConfigPage^.wMaskBtPanelLeft:=16#1F;
ptrConfigPage^.wMaskBtPanelRight:=16#1E0;
ptrConfigPage^.wMaskFunctionPanel:=16#2B;
(* Navigation panel restriction *)
ptrConfigPage^.wMaskTouchScreenNavPanel:=16#27;
(* Active machine movement mask *)
ptrConfigPage^.wMaskActiveMachineBtPanelLeft:=16#0;
ptrConfigPage^.wMaskActiveMachineBtPanelRight:=16#0;
ptrConfigPage^.wMaskActiveMachineFunctionPanel:=16#0;
ptrConfigPage^.wMaskActiveMachineNavPanel:=16#27;
(* Button edge action *)
ptrConfigPage^.aiRTrigActionPanelRight[1]:=312;
ptrConfigPage^.aiRTrigActionPanelRight[2]:=310;
ptrConfigPage^.aiRTrigActionPanelRight[3]:=316;
ptrConfigPage^.aiRTrigActionPanelRight[4]:=314;
ptrConfigPage^.aiRTrigActionPanelRight[5]:=0;
ptrConfigPage^.aiFTrigActionPanelRight[1]:=0;
ptrConfigPage^.aiFTrigActionPanelRight[2]:=0;
ptrConfigPage^.aiFTrigActionPanelRight[3]:=301;
ptrConfigPage^.aiFTrigActionPanelRight[4]:=301;
ptrConfigPage^.aiFTrigActionPanelRight[5]:=0;
ptrConfigPage^.aiDelayActionPanelRight[1]:=0;
ptrConfigPage^.aiDelayActionPanelRight[2]:=0;
ptrConfigPage^.aiDelayActionPanelRight[3]:=0;
ptrConfigPage^.aiDelayActionPanelRight[4]:=0;
ptrConfigPage^.aiDelayActionPanelRight[5]:=0;
ptrConfigPage^.aiRTrigActionFunctionPanel[1]:=322;
ptrConfigPage^.aiRTrigActionFunctionPanel[2]:=323;
ptrConfigPage^.aiRTrigActionFunctionPanel[3]:=0;
ptrConfigPage^.aiRTrigActionFunctionPanel[4]:=320;
ptrConfigPage^.aiRTrigActionFunctionPanel[5]:=0;
ptrConfigPage^.aiRTrigActionFunctionPanel[6]:=325;
ptrConfigPage^.aiRTrigActionFunctionPanel[7]:=0;
ptrConfigPage^.aiRTrigActionFunctionPanel[8]:=0;
ptrConfigPage^.aiRTrigActionFunctionPanel[9]:=0;
ptrConfigPage^.aiRTrigActionFunctionPanel[10]:=0;
ptrConfigPage^.aiRTrigActionFunctionPanel[11]:=0;
ptrConfigPage^.aiRTrigActionFunctionPanel[12]:=0;
ptrConfigPage^.aiFTrigActionTouchScreenNavPanel[1]:=10410;
ptrConfigPage^.aiFTrigActionTouchScreenNavPanel[2]:=10420;
ptrConfigPage^.aiFTrigActionTouchScreenNavPanel[3]:=10430;
ptrConfigPage^.aiFTrigActionTouchScreenNavPanel[4]:=0;
ptrConfigPage^.aiFTrigActionTouchScreenNavPanel[5]:=0;
ptrConfigPage^.aiFTrigActionTouchScreenNavPanel[6]:=10460;
ptrConfigPage^.xMaskBtStart:=TRUE;
ptrConfigPage^.xMaskBtStop:=TRUE;
END_ACTION
ACTION Page_420_WorkStation_ToolDia:
(* QVis page 420, Tool Diameter *)
iIndexPage:=420;
iPageNumber:=iPageNumber+1;
T_Visu.T_PageIndex[iIndexPage].iIndexConfigPage:=iPageNumber;
ptrConfigPage:=ADR(T_Visu.T_ConfigPage[T_Visu.T_PageIndex[iIndexPage].iIndexConfigPage]);
ptrConfigPage^.sName:='Tool Diameter';
ptrConfigPage^.wMaskBtPanelLeft:=16#1F;
ptrConfigPage^.wMaskBtPanelRight:=16#0;
ptrConfigPage^.wMaskFunctionPanel:=16#EF;
(* Navigation panel restriction *)
ptrConfigPage^.wMaskTouchScreenNavPanel:=16#27;
(* Active machine movement mask *)
ptrConfigPage^.wMaskActiveMachineBtPanelLeft:=16#0;
ptrConfigPage^.wMaskActiveMachineBtPanelRight:=16#0;
ptrConfigPage^.wMaskActiveMachineFunctionPanel:=16#0;
ptrConfigPage^.wMaskActiveMachineNavPanel:=16#27;
(* Button edge action *)
ptrConfigPage^.aiRTrigActionPanelRight[1]:=0;
ptrConfigPage^.aiRTrigActionPanelRight[2]:=0;
ptrConfigPage^.aiRTrigActionPanelRight[3]:=0;
ptrConfigPage^.aiRTrigActionPanelRight[4]:=0;
ptrConfigPage^.aiRTrigActionPanelRight[5]:=0;
ptrConfigPage^.aiFTrigActionPanelRight[1]:=0;
ptrConfigPage^.aiFTrigActionPanelRight[2]:=0;
ptrConfigPage^.aiFTrigActionPanelRight[3]:=0;
ptrConfigPage^.aiFTrigActionPanelRight[4]:=0;
ptrConfigPage^.aiFTrigActionPanelRight[5]:=0;
ptrConfigPage^.aiDelayActionPanelRight[1]:=0;
ptrConfigPage^.aiDelayActionPanelRight[2]:=0;
ptrConfigPage^.aiDelayActionPanelRight[3]:=0;
ptrConfigPage^.aiDelayActionPanelRight[4]:=0;
ptrConfigPage^.aiDelayActionPanelRight[5]:=0;
ptrConfigPage^.aiRTrigActionFunctionPanel[1]:=110;
ptrConfigPage^.aiRTrigActionFunctionPanel[2]:=111;
ptrConfigPage^.aiRTrigActionFunctionPanel[3]:=114;
ptrConfigPage^.aiRTrigActionFunctionPanel[4]:=115;
ptrConfigPage^.aiRTrigActionFunctionPanel[5]:=0;
ptrConfigPage^.aiRTrigActionFunctionPanel[6]:=116;
ptrConfigPage^.aiRTrigActionFunctionPanel[7]:=112;
ptrConfigPage^.aiRTrigActionFunctionPanel[8]:=113;
ptrConfigPage^.aiRTrigActionFunctionPanel[9]:=0;
ptrConfigPage^.aiRTrigActionFunctionPanel[10]:=0;
ptrConfigPage^.aiRTrigActionFunctionPanel[11]:=0;
ptrConfigPage^.aiRTrigActionFunctionPanel[12]:=0;
ptrConfigPage^.aiFTrigActionTouchScreenNavPanel[1]:=10410;
ptrConfigPage^.aiFTrigActionTouchScreenNavPanel[2]:=10420;
ptrConfigPage^.aiFTrigActionTouchScreenNavPanel[3]:=10430;
ptrConfigPage^.aiFTrigActionTouchScreenNavPanel[4]:=0;
ptrConfigPage^.aiFTrigActionTouchScreenNavPanel[5]:=0;
ptrConfigPage^.aiFTrigActionTouchScreenNavPanel[6]:=10460;
ptrConfigPage^.xMaskBtStart:=FALSE;
ptrConfigPage^.xMaskBtStop:=TRUE;
END_ACTION
ACTION Page_430_WorkStation_Prism:
(* QVis page 430, Prism *)
iIndexPage:=430;
iPageNumber:=iPageNumber+1;
T_Visu.T_PageIndex[iIndexPage].iIndexConfigPage:=iPageNumber;
ptrConfigPage:=ADR(T_Visu.T_ConfigPage[T_Visu.T_PageIndex[iIndexPage].iIndexConfigPage]);
ptrConfigPage^.sName:='Prism';
ptrConfigPage^.wMaskBtPanelLeft:=16#1F;
ptrConfigPage^.wMaskBtPanelRight:=16#0;
ptrConfigPage^.wMaskFunctionPanel:=16#3F;
(* Navigation panel restriction *)
ptrConfigPage^.wMaskTouchScreenNavPanel:=16#27;
(* Active machine movement mask *)
ptrConfigPage^.wMaskActiveMachineBtPanelLeft:=16#0;
ptrConfigPage^.wMaskActiveMachineBtPanelRight:=16#0;
ptrConfigPage^.wMaskActiveMachineFunctionPanel:=16#0;
ptrConfigPage^.wMaskActiveMachineNavPanel:=16#27;
(* Button edge action *)
ptrConfigPage^.aiRTrigActionPanelRight[1]:=0;
ptrConfigPage^.aiRTrigActionPanelRight[2]:=0;
ptrConfigPage^.aiRTrigActionPanelRight[3]:=0;
ptrConfigPage^.aiRTrigActionPanelRight[4]:=0;
ptrConfigPage^.aiRTrigActionPanelRight[5]:=0;
ptrConfigPage^.aiFTrigActionPanelRight[1]:=0;
ptrConfigPage^.aiFTrigActionPanelRight[2]:=0;
ptrConfigPage^.aiFTrigActionPanelRight[3]:=0;
ptrConfigPage^.aiFTrigActionPanelRight[4]:=0;
ptrConfigPage^.aiFTrigActionPanelRight[5]:=0;
ptrConfigPage^.aiDelayActionPanelRight[1]:=0;
ptrConfigPage^.aiDelayActionPanelRight[2]:=0;
ptrConfigPage^.aiDelayActionPanelRight[3]:=0;
ptrConfigPage^.aiDelayActionPanelRight[4]:=0;
ptrConfigPage^.aiDelayActionPanelRight[5]:=0;
ptrConfigPage^.aiRTrigActionFunctionPanel[1]:=120;
ptrConfigPage^.aiRTrigActionFunctionPanel[2]:=115;
ptrConfigPage^.aiRTrigActionFunctionPanel[3]:=0;
ptrConfigPage^.aiRTrigActionFunctionPanel[4]:=0;
ptrConfigPage^.aiRTrigActionFunctionPanel[5]:=0;
ptrConfigPage^.aiRTrigActionFunctionPanel[6]:=1005;
ptrConfigPage^.aiRTrigActionFunctionPanel[7]:=0;
ptrConfigPage^.aiRTrigActionFunctionPanel[8]:=0;
ptrConfigPage^.aiRTrigActionFunctionPanel[9]:=0;
ptrConfigPage^.aiRTrigActionFunctionPanel[10]:=0;
ptrConfigPage^.aiRTrigActionFunctionPanel[11]:=0;
ptrConfigPage^.aiRTrigActionFunctionPanel[12]:=0;
ptrConfigPage^.aiFTrigActionTouchScreenNavPanel[1]:=10410;
ptrConfigPage^.aiFTrigActionTouchScreenNavPanel[2]:=10420;
ptrConfigPage^.aiFTrigActionTouchScreenNavPanel[3]:=10430;
ptrConfigPage^.aiFTrigActionTouchScreenNavPanel[4]:=0;
ptrConfigPage^.aiFTrigActionTouchScreenNavPanel[5]:=0;
ptrConfigPage^.aiFTrigActionTouchScreenNavPanel[6]:=10460;
ptrConfigPage^.xMaskBtStart:=FALSE;
ptrConfigPage^.xMaskBtStop:=TRUE;
END_ACTION
ACTION Page_460_WorkStation_ErrorList:
(* QVis page 460, Error List *)
iIndexPage:=460;
iPageNumber:=iPageNumber+1;
T_Visu.T_PageIndex[iIndexPage].iIndexConfigPage:=iPageNumber;
ptrConfigPage:=ADR(T_Visu.T_ConfigPage[T_Visu.T_PageIndex[iIndexPage].iIndexConfigPage]);
ptrConfigPage^.sName:='Error List';
ptrConfigPage^.wMaskBtPanelLeft:=16#1F;
ptrConfigPage^.wMaskBtPanelRight:=16#60;
ptrConfigPage^.wMaskFunctionPanel:=16#0;
(* Navigation panel restriction *)
ptrConfigPage^.wMaskTouchScreenNavPanel:=16#27;
(* Active machine movement mask *)
ptrConfigPage^.wMaskActiveMachineBtPanelLeft:=16#0;
ptrConfigPage^.wMaskActiveMachineBtPanelRight:=16#60;
ptrConfigPage^.wMaskActiveMachineFunctionPanel:=16#0;
ptrConfigPage^.wMaskActiveMachineNavPanel:=16#27;
(* Button edge action *)
ptrConfigPage^.aiRTrigActionPanelRight[1]:=99;
ptrConfigPage^.aiRTrigActionPanelRight[2]:=20;
ptrConfigPage^.aiRTrigActionPanelRight[3]:=0;
ptrConfigPage^.aiRTrigActionPanelRight[4]:=0;
ptrConfigPage^.aiRTrigActionPanelRight[5]:=0;
ptrConfigPage^.aiFTrigActionPanelRight[1]:=0;
ptrConfigPage^.aiFTrigActionPanelRight[2]:=0;
ptrConfigPage^.aiFTrigActionPanelRight[3]:=0;
ptrConfigPage^.aiFTrigActionPanelRight[4]:=0;
ptrConfigPage^.aiFTrigActionPanelRight[5]:=0;
ptrConfigPage^.aiDelayActionPanelRight[1]:=0;
ptrConfigPage^.aiDelayActionPanelRight[2]:=0;
ptrConfigPage^.aiDelayActionPanelRight[3]:=0;
ptrConfigPage^.aiDelayActionPanelRight[4]:=0;
ptrConfigPage^.aiDelayActionPanelRight[5]:=0;
ptrConfigPage^.aiRTrigActionFunctionPanel[1]:=0;
ptrConfigPage^.aiRTrigActionFunctionPanel[2]:=0;
ptrConfigPage^.aiRTrigActionFunctionPanel[3]:=0;
ptrConfigPage^.aiRTrigActionFunctionPanel[4]:=0;
ptrConfigPage^.aiRTrigActionFunctionPanel[5]:=0;
ptrConfigPage^.aiRTrigActionFunctionPanel[6]:=0;
ptrConfigPage^.aiRTrigActionFunctionPanel[7]:=0;
ptrConfigPage^.aiRTrigActionFunctionPanel[8]:=0;
ptrConfigPage^.aiRTrigActionFunctionPanel[9]:=0;
ptrConfigPage^.aiRTrigActionFunctionPanel[10]:=0;
ptrConfigPage^.aiRTrigActionFunctionPanel[11]:=0;
ptrConfigPage^.aiRTrigActionFunctionPanel[12]:=0;
ptrConfigPage^.aiFTrigActionTouchScreenNavPanel[1]:=10410;
ptrConfigPage^.aiFTrigActionTouchScreenNavPanel[2]:=10420;
ptrConfigPage^.aiFTrigActionTouchScreenNavPanel[3]:=10430;
ptrConfigPage^.aiFTrigActionTouchScreenNavPanel[4]:=0;
ptrConfigPage^.aiFTrigActionTouchScreenNavPanel[5]:=0;
ptrConfigPage^.aiFTrigActionTouchScreenNavPanel[6]:=10460;
ptrConfigPage^.xMaskBtStart:=FALSE;
ptrConfigPage^.xMaskBtStop:=TRUE;
END_ACTION
ACTION Page_470_WorkStation_Parameter3:
(* QVis page 470, Parameter Grind Axis *)
iIndexPage:=470;
iPageNumber:=iPageNumber+1;
T_Visu.T_PageIndex[iIndexPage].iIndexConfigPage:=iPageNumber;
ptrConfigPage:=ADR(T_Visu.T_ConfigPage[T_Visu.T_PageIndex[iIndexPage].iIndexConfigPage]);
ptrConfigPage^.sName:='Parameter Grind Axis';
ptrConfigPage^.wMaskBtPanelLeft:=16#1F;
ptrConfigPage^.wMaskBtPanelRight:=16#200;
ptrConfigPage^.wMaskFunctionPanel:=16#0;
(* Navigation panel restriction *)
ptrConfigPage^.wMaskTouchScreenNavPanel:=16#27;
(* Active machine movement mask *)
ptrConfigPage^.wMaskActiveMachineBtPanelLeft:=16#0;
ptrConfigPage^.wMaskActiveMachineBtPanelRight:=16#0;
ptrConfigPage^.wMaskActiveMachineFunctionPanel:=16#0;
ptrConfigPage^.wMaskActiveMachineNavPanel:=16#27;
(* Button edge action *)
ptrConfigPage^.aiRTrigActionPanelRight[1]:=0;
ptrConfigPage^.aiRTrigActionPanelRight[2]:=0;
ptrConfigPage^.aiRTrigActionPanelRight[3]:=0;
ptrConfigPage^.aiRTrigActionPanelRight[4]:=0;
ptrConfigPage^.aiRTrigActionPanelRight[5]:=1006;
ptrConfigPage^.aiFTrigActionPanelRight[1]:=0;
ptrConfigPage^.aiFTrigActionPanelRight[2]:=0;
ptrConfigPage^.aiFTrigActionPanelRight[3]:=0;
ptrConfigPage^.aiFTrigActionPanelRight[4]:=0;
ptrConfigPage^.aiFTrigActionPanelRight[5]:=0;
ptrConfigPage^.aiDelayActionPanelRight[1]:=0;
ptrConfigPage^.aiDelayActionPanelRight[2]:=0;
ptrConfigPage^.aiDelayActionPanelRight[3]:=0;
ptrConfigPage^.aiDelayActionPanelRight[4]:=0;
ptrConfigPage^.aiDelayActionPanelRight[5]:=0;
ptrConfigPage^.aiRTrigActionFunctionPanel[1]:=0;
ptrConfigPage^.aiRTrigActionFunctionPanel[2]:=0;
ptrConfigPage^.aiRTrigActionFunctionPanel[3]:=0;
ptrConfigPage^.aiRTrigActionFunctionPanel[4]:=0;
ptrConfigPage^.aiRTrigActionFunctionPanel[5]:=0;
ptrConfigPage^.aiRTrigActionFunctionPanel[6]:=0;
ptrConfigPage^.aiRTrigActionFunctionPanel[7]:=0;
ptrConfigPage^.aiRTrigActionFunctionPanel[8]:=0;
ptrConfigPage^.aiRTrigActionFunctionPanel[9]:=0;
ptrConfigPage^.aiRTrigActionFunctionPanel[10]:=0;
ptrConfigPage^.aiRTrigActionFunctionPanel[11]:=0;
ptrConfigPage^.aiRTrigActionFunctionPanel[12]:=0;
ptrConfigPage^.aiFTrigActionTouchScreenNavPanel[1]:=10410;
ptrConfigPage^.aiFTrigActionTouchScreenNavPanel[2]:=10420;
ptrConfigPage^.aiFTrigActionTouchScreenNavPanel[3]:=10430;
ptrConfigPage^.aiFTrigActionTouchScreenNavPanel[4]:=0;
ptrConfigPage^.aiFTrigActionTouchScreenNavPanel[5]:=0;
ptrConfigPage^.aiFTrigActionTouchScreenNavPanel[6]:=10460;
ptrConfigPage^.xMaskBtStart:=FALSE;
ptrConfigPage^.xMaskBtStop:=TRUE;
END_ACTION

(* POU PRG_VISU_LAYER5/FB_VISU/FB_COMPAREPROFILEPROCESSVALUE, ST *)
FUNCTION_BLOCK FB_COMPAREPROFILEPROCESSVALUE
VAR_INPUT
	T_Data_ProcessImageLoadData:ST_RETAIN_DATA_PROCESSIMAGE;	(* Novram parameter structure for the profile value *)
	T_Data_ProcessImageData:ST_RETAIN_DATA_PROCESSIMAGE;		(* Novram parametre structure for the process parameter *)
	xMicroRodActive: BOOL;											(* choice of the machine MicroWire or MicroRod *)
END_VAR
VAR_OUTPUT
	xProcessValueModified:BOOL;										(* TRUE=Profile parameter and process parameter are not the same, FALSE=both are same *)
END_VAR
VAR_IN_OUT
END_VAR
VAR
(* variable *)
	xFirstExecution:BOOL;
END_VAR
(****************************************************************************************************************************************************)
(***  This Functionblock check if the parameter of the loaded profile ar the same as the parameter of the process parameter   ***)
(****************************************************************************************************************************************************)
(* First execution *)
	IF NOT xFirstExecution THEN
		xProcessValueModified:=FALSE;
		(* confirm execution *)
		xFirstExecution:=TRUE;
	END_IF

(* compare value *)
	xProcessValueModified:=FALSE;

	(* value *)
	IF T_Data_ProcessImageLoadData.T_GeometryPara.arStartDiameter[1] <> T_Data_ProcessImageData.T_GeometryPara.arStartDiameter[1] THEN xProcessValueModified:=TRUE; RETURN; END_IF
	IF T_Data_ProcessImageLoadData.T_GeometryPara.arEndDiameter[1] <> T_Data_ProcessImageData.T_GeometryPara.arEndDiameter[1] THEN xProcessValueModified:=TRUE; RETURN; END_IF
	IF T_Data_ProcessImageLoadData.T_GeometryPara.arSectionLength[1] <> T_Data_ProcessImageData.T_GeometryPara.arSectionLength[1] THEN xProcessValueModified:=TRUE; RETURN; END_IF
	IF T_Data_ProcessImageLoadData.T_GeometryPara.arSectionPitch[1] <> T_Data_ProcessImageData.T_GeometryPara.arSectionPitch[1] THEN xProcessValueModified:=TRUE; RETURN; END_IF
	IF T_Data_ProcessImageLoadData.T_GeometryPara.axActiveSection[1] <> T_Data_ProcessImageData.T_GeometryPara.axActiveSection[1] THEN xProcessValueModified:=TRUE; RETURN; END_IF

	IF T_Data_ProcessImageLoadData.T_GeometryPara.arStartDiameter[2] <> T_Data_ProcessImageData.T_GeometryPara.arStartDiameter[2] THEN xProcessValueModified:=TRUE; RETURN; END_IF
	IF T_Data_ProcessImageLoadData.T_GeometryPara.arEndDiameter[2] <> T_Data_ProcessImageData.T_GeometryPara.arEndDiameter[2] THEN xProcessValueModified:=TRUE; RETURN; END_IF
	IF T_Data_ProcessImageLoadData.T_GeometryPara.arSectionLength[2] <> T_Data_ProcessImageData.T_GeometryPara.arSectionLength[2] THEN xProcessValueModified:=TRUE; RETURN; END_IF
	IF T_Data_ProcessImageLoadData.T_GeometryPara.arSectionPitch[2] <> T_Data_ProcessImageData.T_GeometryPara.arSectionPitch[2] THEN xProcessValueModified:=TRUE; RETURN; END_IF
	IF T_Data_ProcessImageLoadData.T_GeometryPara.axActiveSection[2] <> T_Data_ProcessImageData.T_GeometryPara.axActiveSection[2] THEN xProcessValueModified:=TRUE; RETURN; END_IF

	IF T_Data_ProcessImageLoadData.T_GeometryPara.arStartDiameter[3] <> T_Data_ProcessImageData.T_GeometryPara.arStartDiameter[3] THEN xProcessValueModified:=TRUE; RETURN; END_IF
	IF T_Data_ProcessImageLoadData.T_GeometryPara.arEndDiameter[3] <> T_Data_ProcessImageData.T_GeometryPara.arEndDiameter[3] THEN xProcessValueModified:=TRUE; RETURN; END_IF
	IF T_Data_ProcessImageLoadData.T_GeometryPara.arSectionLength[3] <> T_Data_ProcessImageData.T_GeometryPara.arSectionLength[3] THEN xProcessValueModified:=TRUE; RETURN; END_IF
	IF T_Data_ProcessImageLoadData.T_GeometryPara.arSectionPitch[3] <> T_Data_ProcessImageData.T_GeometryPara.arSectionPitch[3] THEN xProcessValueModified:=TRUE; RETURN; END_IF
	IF T_Data_ProcessImageLoadData.T_GeometryPara.axActiveSection[3] <> T_Data_ProcessImageData.T_GeometryPara.axActiveSection[3] THEN xProcessValueModified:=TRUE; RETURN; END_IF

	IF T_Data_ProcessImageLoadData.T_GeometryPara.arStartDiameter[4] <> T_Data_ProcessImageData.T_GeometryPara.arStartDiameter[4] THEN xProcessValueModified:=TRUE; RETURN; END_IF
	IF T_Data_ProcessImageLoadData.T_GeometryPara.arEndDiameter[4] <> T_Data_ProcessImageData.T_GeometryPara.arEndDiameter[4] THEN xProcessValueModified:=TRUE; RETURN; END_IF
	IF T_Data_ProcessImageLoadData.T_GeometryPara.arSectionLength[4] <> T_Data_ProcessImageData.T_GeometryPara.arSectionLength[4] THEN xProcessValueModified:=TRUE; RETURN; END_IF
	IF T_Data_ProcessImageLoadData.T_GeometryPara.arSectionPitch[4] <> T_Data_ProcessImageData.T_GeometryPara.arSectionPitch[4] THEN xProcessValueModified:=TRUE; RETURN; END_IF
	IF T_Data_ProcessImageLoadData.T_GeometryPara.axActiveSection[4] <> T_Data_ProcessImageData.T_GeometryPara.axActiveSection[4] THEN xProcessValueModified:=TRUE; RETURN; END_IF
(*09.12.2022: SOA *)
	IF T_Data_ProcessImageLoadData.T_GeometryPara.arStartDiameter[5] <> T_Data_ProcessImageData.T_GeometryPara.arStartDiameter[5] THEN xProcessValueModified:=TRUE; RETURN; END_IF
	IF T_Data_ProcessImageLoadData.T_GeometryPara.arEndDiameter[5] <> T_Data_ProcessImageData.T_GeometryPara.arEndDiameter[5] THEN xProcessValueModified:=TRUE; RETURN; END_IF
	IF T_Data_ProcessImageLoadData.T_GeometryPara.arSectionLength[5] <> T_Data_ProcessImageData.T_GeometryPara.arSectionLength[5] THEN xProcessValueModified:=TRUE; RETURN; END_IF
	IF T_Data_ProcessImageLoadData.T_GeometryPara.arSectionPitch[5] <> T_Data_ProcessImageData.T_GeometryPara.arSectionPitch[5] THEN xProcessValueModified:=TRUE; RETURN; END_IF
	IF T_Data_ProcessImageLoadData.T_GeometryPara.axActiveSection[5] <> T_Data_ProcessImageData.T_GeometryPara.axActiveSection[5] THEN xProcessValueModified:=TRUE; RETURN; END_IF

